// TwinCAT 3 PLC project EngineeringToolbox
// Title: EngineeringToolbox
// Company: Beckhoff Electronics Mfg
// Author: Daniel Schlingmann
// ProjectVersion: 3.1.2.2
// Description: Engineering Toolbox Library The library is provided "as-is" for TwinCAT3.1 by the Beckhoff Industry Management for Electronics Manufacturing. Please check the function "DisclaimerStatement : WSTRING[1500]" in additon to the following disclaimer: THE SOFTWARE IS PROVIDED "AS IS", WITHOUT WARRANTY OF ANY KIND, EXPRESS OR IMPLIED, INCLUDING BUT NOT LIMITED TO THE WARRANTIES OF MERCHANTABILITY, FITNESS FOR A PARTICULAR PURPOSE AND NONINFRINGEMENT. IN NO EVENT SHALL THE AUTHORS OR COPYRIGHT HOLDERS BE LIABLE FOR ANY CLAIM, DAMAGES OR OTHER LIABILITY, WHETHER IN AN ACTION OF CONTRACT, TORT OR OTHERWISE, ARISING FROM, OUT OF OR IN CONNECTION WITH THE SOFTWARE OR THE USE OR OTHER DEALINGS IN THE SOFTWARE.
// ProgramVersion: 3.1.4022.7
// libraries:
//   Tc2_Drive, * (Beckhoff Automation GmbH)
//   Tc2_EtherCAT, * (Beckhoff Automation GmbH)
//   Tc2_IoFunctions, * (Beckhoff Automation GmbH)
//   Tc2_Math, * (Beckhoff Automation GmbH)
//   Tc2_MC2, * (Beckhoff Automation GmbH)
//   Tc2_MC2_Camming, * (Beckhoff Automation GmbH)
//   Tc2_MC2_Drive, * (Beckhoff Automation GmbH)
//   Tc2_MC2_FlyingSaw, * (Beckhoff Automation GmbH)
//   Tc2_MDP, * (Beckhoff Automation GmbH)
//   Tc2_ModbusRTU, * (Beckhoff Automation GmbH)
//   Tc2_ModbusSrv, * (Beckhoff Automation GmbH)
//   Tc2_NC, * (Beckhoff Automation GmbH)
//   Tc2_NCI, * (Beckhoff Automation GmbH)
//   Tc2_NcKinematicTransformation, * (Beckhoff Automation GmbH)
//   Tc2_PlcInterpolation, * (Beckhoff Automation GmbH)
//   Tc2_SerialCom, * (Beckhoff Automation GmbH)
//   Tc2_Smtp, * (Beckhoff Automation GmbH)
//   Tc2_Standard, * (Beckhoff Automation GmbH)
//   Tc2_SUPS, * (Beckhoff Automation GmbH)
//   Tc2_System, * (Beckhoff Automation GmbH)
//   Tc2_TcpIp, * (Beckhoff Automation GmbH)
//   Tc2_Utilities, * (Beckhoff Automation GmbH)
//   Tc2_XmlDataSrv, * (Beckhoff Automation GmbH)
//   Tc3_Module, * (Beckhoff Automation GmbH)
//   Tc2_BackupRestoreEL6900,newest,Beckhoff Automation GmbH
// project tree:
//   GVLs/ Gvl.TcGVL (not stored), PARAM.TcGVL (not stored)
//   POUs/BoundsCheck/ boundsError.TcPOU (not stored), boundsOK.TcPOU (not stored), checkBounds.TcPOU (not stored), CheckBoundsInfo.TcPOU (not stored)
//   POUs/Connectivity/ADS/ AdsDataExchange.TcPOU
//   POUs/Connectivity/ Ipv4Addr_TO_UDINT.TcPOU, U_DEVICE_COM_CACHE.TcDUT (not stored), U_IPv4Addr.TcDUT (not stored), isValidIPv4Addr.TcPOU (not stored)
//   POUs/Connectivity/TF6310-TcpServer/DeviceCom/ TCPDeviceCom_SendRecBytes.TcPOU (not stored), TCPDeviceCom_SendRecString.TcPOU (not stored)
//   POUs/Connectivity/TF6340-SerialCom/ComPortDeviceCom/ ComPortDeviceCom_BufferHandle.TcPOU (not stored), ComPortDeviceCom_SendRecBytes.TcPOU (not stored), ComPortDeviceCom_SendRecString.TcPOU (not stored), ComPortEL6x22BEasyConnect.TcPOU (not stored)
//   POUs/Connectivity/TF6340-SerialCom/ComPortBasic/ ComPortBackground.TcPOU (not stored), ComPortSendRec.TcPOU (not stored)
//   POUs/Connectivity/TF625x-Modbus/Master/TF6250-ModbusTcpServer/TCP/ ModbusTcpMaster.TcPOU (not stored)
//   POUs/Connectivity/TF625x-Modbus/Master/TF6250-ModbusTcpServer/UDP/ ModbusUdpMaster.TcPOU
//   POUs/Connectivity/TF625x-Modbus/Master/TF6255-ModbusRtu/ ModbusRtuMaster22B.TcPOU (not stored), ModbusRtuMaster5B.TcPOU (not stored), ModbusRtuMasterPC.TcPOU
//   POUs/Connectivity/TF625x-Modbus/Master/_Components/ ModbusJob.TcPOU (not stored), ModbusSlaveCom.TcPOU (not stored)
//   POUs/Connectivity/TF625x-Modbus/Slave/ ModbusSlaveBase.TcPOU (not stored)
//   POUs/Connectivity/TF6310-TcpServer/TcpBasic/ TCPSendRecCtrl.TcPOU (not stored), TCPConnectionCtrl.TcPOU (not stored), TCPSocketCtrl.TcPOU (not stored)
//   POUs/Connectivity/TF6310-TcpServer/UdpBasic/ UDPSendRecCtrl.TcPOU, UDPServerCtrl.TcPOU (not stored), UDPSocketCtrl.TcPOU (not stored)
//   POUs/ControllerTools/ AverageFilter.TcPOU (not stored), PIDController.TcPOU (not stored), PT1Filter.TcPOU, signum.TcPOU (not stored), SlewRateLimitter.TcPOU (not stored), SlidingAverageExt.TcPOU (not stored), SlidingAverage.TcPOU (not stored), ThreePointController.TcPOU (not stored)
//   POUs/DataBuffer/ DoubleBuffer.TcPOU (not stored), Quicksort.TcPOU (not stored)
//   POUs/DataBuffer/Fifo/ Fifo.TcPOU (not stored), FifoExt.TcPOU (not stored), FifoLRealSimple.TcPOU (not stored), FifoBase.TcPOU (not stored)
//   POUs/DataBuffer/Ringbuffer/ RingbufferBase.TcPOU (not stored), Ringbuffer.TcPOU (not stored), RingbufferCharSimple.TcPOU (not stored), RingbufferExt.TcPOU, RingbufferByteSimple.TcPOU (not stored), RingbufferLRealSimple.TcPOU (not stored)
//   POUs/EventLogger/ EventsWriteToLogbook.TcPOU (not stored), EVENT_HANDLING_CONFIG.TcDUT (not stored), getEventClassPriority.TcPOU, getEventClassText.TcPOU (not stored), SOURCE_ID.TcDUT (not stored)
//   POUs/EventLogger/ReadEvents/ EventlogRead.TcPOU (not stored), EVENTLOG_READ_DATA.TcDUT (not stored), EVENTLOG_READ_HANDLEINFO.TcDUT (not stored), EVENTLOG_READ_STREAM.TcDUT, EVENTLOG_READ_STREAM_DATA_RAW.TcDUT (not stored), EVENTLOG_READ_STREAM_DATA_RAW_EX.TcDUT (not stored)
//   POUs/EventLogger/TriggerEvents/ EventHandling.TcPOU (not stored), EventHandlingGrp10.TcPOU (not stored), EventHandlingGrp25.TcPOU (not stored), EventHandlingGrp50.TcPOU (not stored), EventHandlingGrpCustomized.TcPOU (not stored), EventHandlingConfirmIsReq.TcPOU (not stored), EventHandlingStatisticInfo.TcPOU (not stored)
//   POUs/Fieldbus/CANopen/ CANopenMasterDiag.TcPOU (not stored), CANopenMasterIO.TcPOU (not stored)
//   POUs/Fieldbus/EAP/ EAP_PUB_SUB_IO.TcPOU (not stored), EAP_DEVICE_IO.TcPOU (not stored), EAP_PUB_VAR.TcPOU (not stored), EAP_SUB_VAR.TcPOU (not stored)
//   POUs/Fieldbus/EtherCAT/ EcCoEReadNewestDiagMsg.TcPOU (not stored), EcDiagBase.TcPOU (not stored), EcDiagBase_wEvents.TcPOU (not stored)
//   POUs/Fieldbus/EtherCAT/_Components/ EcMasterIO.TcPOU (not stored), EcMasterSupervisor.TcPOU (not stored), EcSlavesDiag.TcPOU (not stored), EcSlaveSupervisor.TcPOU (not stored), EC_MASTER_DEVICE_STATE.TcDUT (not stored), EC_SLAVE_DIAG_INFO_DATA.TcDUT (not stored)
//   POUs/Fieldbus/Profibus/ ProfibusMasterDiag.TcPOU, ProfibusMasterIO.TcPOU (not stored)
//   POUs/Fieldbus/Profinet/ ProfinetControllerIO.TcPOU (not stored), ProfinetControllerIO_wEvents.TcPOU, ProfinetDeviceIO.TcPOU
//   POUs/FileHandling/Basic/ FileHandling.TcPOU (not stored), ReadDirSimple.TcPOU (not stored), ReadDirSimpleExt.TcPOU (not stored)
//   POUs/FileHandling/TF6421-XmlServer/ XmlReadWrite.TcPOU (not stored), XmlReadWriteWithBackupFile.TcPOU (not stored)
//   POUs/IO/Analog/ AnalogIn.TcPOU, AnalogIn32.TcPOU, AnalogInELMBase.TcPOU (not stored), AnalogInELMSingleSampleDINT.TcPOU (not stored), AnalogInELMSingleSampleREAL.TcPOU (not stored), AnalogInREAL.TcPOU (not stored), AnalogOut.TcPOU
//   POUs/IO/ BlowOffSensors.TcPOU (not stored), Button.TcPOU (not stored), ButtonExt.TcPOU, Fuse.TcPOU (not stored), InOut.TcPOU (not stored), InOutExt.TcPOU, Input.TcPOU (not stored), Output.TcPOU (not stored)
//   POUs/IO/Cylinder/ Cylinder.TcPOU (not stored), CylinderExt.TcPOU (not stored), CylinderType4.TcPOU (not stored), I_Cylinder.TcIO (not stored)
//   POUs/IO/Drives/ AxDriveBase.TcPOU (not stored), AxDriveGetRef.TcPOU (not stored), I_AxDriveBase.TcIO (not stored)
//   POUs/IO/Drives/CoE/ AxDriveCoE.TcPOU (not stored), AxDriveCoE_wEvents.TcPOU (not stored), CiA_DS402Controlword.TcPOU (not stored), CiA_DS402Statusword.TcPOU (not stored), eCiA_DS402_CONTROL_CMD.TcDUT (not stored), eCiA_DS402_STATUS_STATE.TcDUT
//   POUs/IO/Drives/CoE/EL72xx/ AxDriveCoE_EL72xxParam.TcPOU (not stored), CiA_DS402StatuswordEx7xxx.TcPOU (not stored)
//   POUs/IO/Drives/DC/Ey73xx/ AxDriveDC.TcPOU (not stored), AxDriveDC_wEvents.TcPOU (not stored)
//   POUs/IO/Drives/SoE/ AxDriveSoE_Ax5000CommutationCalib.TcPOU (not stored), AxDriveSoE_Ax5000CalcPower.TcPOU (not stored), AxDriveSoE_Ax5000SwitchParamSet.TcPOU (not stored), Ax580x.TcPOU (not stored), AxDriveSoE_Ax5000.TcPOU (not stored), AxDriveSoE_Ax5000Param.TcPOU (not stored), AxDriveSoE_Ax5000wEvents.TcPOU (not stored), AxDriveSoE_Rexroth.TcPOU (not stored)
//   POUs/IO/Drives/SoE/Ax5000ParamSTRUCTs/P/ AX5000_P_0001.TcDUT (not stored), AX5000_P_0002.TcDUT (not stored), AX5000_P_0003.TcDUT (not stored), AX5000_P_0004.TcDUT (not stored), AX5000_P_0009.TcDUT (not stored), AX5000_P_0010.TcDUT (not stored), AX5000_P_0020.TcDUT (not stored), AX5000_P_0021.TcDUT (not stored), AX5000_P_0040.TcDUT (not stored), AX5000_P_0050.TcDUT (not stored), AX5000_P_0051.TcDUT (not stored), AX5000_P_0052.TcDUT (not stored), AX5000_P_0053.TcDUT (not stored), AX5000_P_0054.TcDUT (not stored), AX5000_P_0055.TcDUT (not stored), AX5000_P_0056.TcDUT (not stored), AX5000_P_0057.TcDUT (not stored), AX5000_P_0058.TcDUT, AX5000_P_0059.TcDUT (not stored), AX5000_P_0060.TcDUT (not stored), AX5000_P_0061.TcDUT (not stored), AX5000_P_0062.TcDUT (not stored), AX5000_P_0063.TcDUT, AX5000_P_0064.TcDUT (not stored), AX5000_P_0065.TcDUT (not stored), AX5000_P_0066.TcDUT (not stored), AX5000_P_0067.TcDUT (not stored), AX5000_P_0068.TcDUT (not stored), AX5000_P_0069.TcDUT, AX5000_P_0070.TcDUT (not stored), AX5000_P_0071.TcDUT, AX5000_P_0072.TcDUT, AX5000_P_0073.TcDUT (not stored), AX5000_P_0074.TcDUT (not stored), AX5000_P_0075.TcDUT (not stored), AX5000_P_0076.TcDUT (not stored), AX5000_P_0077.TcDUT (not stored), AX5000_P_0078.TcDUT (not stored), AX5000_P_0088.TcDUT (not stored), AX5000_P_0089.TcDUT (not stored), AX5000_P_0090.TcDUT (not stored), AX5000_P_0091.TcDUT (not stored), AX5000_P_0092.TcDUT (not stored), AX5000_P_0093.TcDUT (not stored), AX5000_P_0096.TcDUT (not stored), AX5000_P_0097.TcDUT (not stored), AX5000_P_0098_beckhoff.TcDUT (not stored), AX5000_P_0098_beckhoff_electrical_data.TcDUT (not stored), AX5000_P_0099.TcDUT (not stored), AX5000_P_0100.TcDUT (not stored), AX5000_P_0101.TcDUT (not stored), AX5000_P_0102.TcDUT (not stored), AX5000_P_0103.TcDUT (not stored), AX5000_P_0104.TcDUT (not stored), AX5000_P_0105.TcDUT (not stored), AX5000_P_0106.TcDUT, AX5000_P_0107.TcDUT (not stored), AX5000_P_0108.TcDUT (not stored), AX5000_P_0109.TcDUT (not stored), AX5000_P_0110.TcDUT (not stored), AX5000_P_0111.TcDUT (not stored), AX5000_P_0112.TcDUT (not stored), AX5000_P_0113.TcDUT (not stored), AX5000_P_0114.TcDUT (not stored), AX5000_P_0115.TcDUT (not stored), AX5000_P_0116.TcDUT (not stored), AX5000_P_0117.TcDUT (not stored), AX5000_P_0118.TcDUT (not stored), AX5000_P_0119.TcDUT (not stored), AX5000_P_0125.TcDUT, AX5000_P_0126.TcDUT (not stored), AX5000_P_0127.TcDUT, AX5000_P_0128.TcDUT (not stored), AX5000_P_0150.TcDUT (not stored), AX5000_P_0151.TcDUT (not stored), AX5000_P_0152.TcDUT (not stored), AX5000_P_0153.TcDUT (not stored), AX5000_P_0154.TcDUT (not stored), AX5000_P_0155.TcDUT (not stored), AX5000_P_0158.TcDUT (not stored), AX5000_P_0159.TcDUT (not stored), AX5000_P_0160.TcDUT (not stored), AX5000_P_0161.TcDUT (not stored), AX5000_P_0162.TcDUT (not stored), AX5000_P_0163.TcDUT (not stored), AX5000_P_0165.TcDUT (not stored), AX5000_P_0166.TcDUT (not stored), AX5000_P_0167.TcDUT (not stored), AX5000_P_0168.TcDUT (not stored), AX5000_P_0169.TcDUT (not stored), AX5000_P_0170.TcDUT, AX5000_P_0171.TcDUT (not stored), AX5000_P_0180.TcDUT (not stored), AX5000_P_0181.TcDUT, AX5000_P_0182.TcDUT (not stored), AX5000_P_0183.TcDUT (not stored), AX5000_P_0184.TcDUT (not stored), AX5000_P_0185.TcDUT (not stored), AX5000_P_0188.TcDUT (not stored), AX5000_P_0189.TcDUT (not stored), AX5000_P_0192.TcDUT (not stored), AX5000_P_0193.TcDUT (not stored), AX5000_P_0196.TcDUT (not stored), AX5000_P_0198.TcDUT, AX5000_P_0199.TcDUT (not stored), AX5000_P_0200.TcDUT, AX5000_P_0201.TcDUT (not stored), AX5000_P_0202.TcDUT, AX5000_P_0203.TcDUT (not stored), AX5000_P_0204.TcDUT (not stored), AX5000_P_0205.TcDUT (not stored), AX5000_P_0206.TcDUT, AX5000_P_0207.TcDUT, AX5000_P_0208.TcDUT, AX5000_P_0209.TcDUT, AX5000_P_0210.TcDUT (not stored), AX5000_P_0211.TcDUT, AX5000_P_0212.TcDUT (not stored), AX5000_P_0213.TcDUT (not stored), AX5000_P_0214.TcDUT (not stored), AX5000_P_0215.TcDUT (not stored), AX5000_P_0216.TcDUT (not stored), AX5000_P_0217.TcDUT, AX5000_P_0218.TcDUT (not stored), AX5000_P_0219.TcDUT (not stored), AX5000_P_0220.TcDUT (not stored), AX5000_P_0221.TcDUT (not stored), AX5000_P_0250.TcDUT (not stored), AX5000_P_0251.TcDUT (not stored), AX5000_P_0252.TcDUT (not stored), AX5000_P_0253.TcDUT (not stored), AX5000_P_0254.TcDUT, AX5000_P_0255.TcDUT (not stored), AX5000_P_0256.TcDUT (not stored), AX5000_P_0270.TcDUT (not stored), AX5000_P_0271.TcDUT (not stored), AX5000_P_0272.TcDUT (not stored), AX5000_P_0273.TcDUT (not stored), AX5000_P_0274.TcDUT (not stored), AX5000_P_0275.TcDUT (not stored), AX5000_P_0276.TcDUT (not stored), AX5000_P_0277.TcDUT (not stored), AX5000_P_0278.TcDUT (not stored), AX5000_P_0300.TcDUT (not stored), AX5000_P_0301.TcDUT (not stored), AX5000_P_0302.TcDUT, AX5000_P_0303.TcDUT (not stored), AX5000_P_0304.TcDUT (not stored), AX5000_P_0305.TcDUT (not stored), AX5000_P_0306.TcDUT (not stored), AX5000_P_0307.TcDUT (not stored), AX5000_P_0308.TcDUT (not stored), AX5000_P_0309.TcDUT (not stored), AX5000_P_0310.TcDUT (not stored), AX5000_P_0311.TcDUT (not stored), AX5000_P_0312.TcDUT (not stored), AX5000_P_0313.TcDUT (not stored), AX5000_P_0314.TcDUT (not stored), AX5000_P_0315.TcDUT (not stored), AX5000_P_0316.TcDUT (not stored), AX5000_P_0317.TcDUT (not stored), AX5000_P_0320.TcDUT (not stored), AX5000_P_0321.TcDUT (not stored), AX5000_P_0322.TcDUT (not stored), AX5000_P_0323.TcDUT (not stored), AX5000_P_0324.TcDUT (not stored), AX5000_P_0325.TcDUT (not stored), AX5000_P_0326.TcDUT (not stored), AX5000_P_0350.TcDUT (not stored), AX5000_P_0351.TcDUT (not stored), AX5000_P_0352.TcDUT, AX5000_P_0353.TcDUT (not stored), AX5000_P_0354.TcDUT, AX5000_P_0356.TcDUT (not stored), AX5000_P_0360.TcDUT (not stored), AX5000_P_0361.TcDUT (not stored), AX5000_P_0400.TcDUT (not stored), AX5000_P_0401.TcDUT (not stored), AX5000_P_0402.TcDUT (not stored), AX5000_P_0451.TcDUT (not stored), AX5000_P_0452.TcDUT (not stored), AX5000_P_0453.TcDUT (not stored), AX5000_P_0454.TcDUT (not stored), AX5000_P_0455.TcDUT (not stored), AX5000_P_0456.TcDUT (not stored), AX5000_P_0457.TcDUT (not stored), AX5000_P_0458.TcDUT (not stored), AX5000_P_0459.TcDUT (not stored), AX5000_P_0460.TcDUT (not stored), AX5000_P_0461.TcDUT (not stored), AX5000_P_0462.TcDUT (not stored), AX5000_P_0463.TcDUT (not stored), AX5000_P_0464.TcDUT, AX5000_P_0502.TcDUT (not stored), AX5000_P_0503.TcDUT (not stored), AX5000_P_0504.TcDUT (not stored), AX5000_P_0505.TcDUT, AX5000_P_0511.TcDUT (not stored), AX5000_P_0512.TcDUT (not stored), AX5000_P_0513.TcDUT (not stored), AX5000_P_0514.TcDUT, AX5000_P_0515.TcDUT (not stored), AX5000_P_0516.TcDUT, AX5000_P_0517.TcDUT (not stored), AX5000_P_0518.TcDUT (not stored), AX5000_P_0552.TcDUT (not stored), AX5000_P_0553.TcDUT (not stored), AX5000_P_0554.TcDUT (not stored), AX5000_P_0555.TcDUT (not stored), AX5000_P_0556.TcDUT (not stored), AX5000_P_0557.TcDUT, AX5000_P_0558.TcDUT (not stored), AX5000_P_0601.TcDUT (not stored), AX5000_P_0602.TcDUT (not stored), AX5000_P_0610.TcDUT (not stored), AX5000_P_0611.TcDUT (not stored), AX5000_P_0800.TcDUT (not stored), AX5000_P_0801.TcDUT (not stored), AX5000_P_0802.TcDUT (not stored), AX5000_P_0804.TcDUT (not stored), AX5000_P_0805.TcDUT (not stored), AX5000_P_0806.TcDUT (not stored), AX5000_P_0810.TcDUT (not stored), AX5000_P_0811.TcDUT, AX5000_P_0850.TcDUT (not stored), AX5000_P_0851.TcDUT (not stored), AX5000_P_0900.TcDUT, AX5000_P_0901.TcDUT (not stored), AX5000_P_0902.TcDUT (not stored), AX5000_P_0904.TcDUT (not stored), AX5000_P_0905.TcDUT (not stored), AX5000_P_0906.TcDUT (not stored), AX5000_P_0912.TcDUT (not stored), AX5000_P_1000.TcDUT (not stored), AX5000_P_1001.TcDUT (not stored), AX5000_P_1002.TcDUT (not stored), AX5000_P_1003.TcDUT (not stored), AX5000_P_1004.TcDUT (not stored), AX5000_P_1005.TcDUT (not stored), AX5000_P_1006.TcDUT (not stored), AX5000_P_1007.TcDUT (not stored), AX5000_P_1008.TcDUT (not stored), AX5000_P_1009.TcDUT, AX5000_P_1010.TcDUT, AX5000_P_1011.TcDUT (not stored), AX5000_P_1012.TcDUT (not stored), AX5000_P_1020.TcDUT (not stored), AX5000_P_1021.TcDUT (not stored), AX5000_P_1022.TcDUT (not stored), AX5000_P_2000.TcDUT (not stored), AX5000_P_2001.TcDUT (not stored), AX5000_P_2002.TcDUT (not stored)
//   POUs/IO/Drives/SoE/Ax5000ParamSTRUCTs/S/ AX5000_S_0001.TcDUT (not stored), AX5000_S_0002.TcDUT (not stored), AX5000_S_0007.TcDUT (not stored), AX5000_S_0011.TcDUT (not stored), AX5000_S_0012.TcDUT (not stored), AX5000_S_0013.TcDUT (not stored), AX5000_S_0015.TcDUT (not stored), AX5000_S_0016.TcDUT, AX5000_S_0017.TcDUT (not stored), AX5000_S_0018.TcDUT (not stored), AX5000_S_0024.TcDUT, AX5000_S_0029.TcDUT, AX5000_S_0030.TcDUT (not stored), AX5000_S_0031.TcDUT (not stored), AX5000_S_0032.TcDUT, AX5000_S_0033.TcDUT (not stored), AX5000_S_0034.TcDUT (not stored), AX5000_S_0035.TcDUT, AX5000_S_0036.TcDUT, AX5000_S_0037.TcDUT (not stored), AX5000_S_0040.TcDUT (not stored), AX5000_S_0043.TcDUT (not stored), AX5000_S_0044.TcDUT (not stored), AX5000_S_0045.TcDUT (not stored), AX5000_S_0046.TcDUT (not stored), AX5000_S_0047.TcDUT (not stored), AX5000_S_0048.TcDUT (not stored), AX5000_S_0051.TcDUT (not stored), AX5000_S_0053.TcDUT (not stored), AX5000_S_0055.TcDUT, AX5000_S_0076.TcDUT (not stored), AX5000_S_0079.TcDUT (not stored), AX5000_S_0080.TcDUT (not stored), AX5000_S_0081.TcDUT (not stored), AX5000_S_0082.TcDUT, AX5000_S_0083.TcDUT, AX5000_S_0084.TcDUT (not stored), AX5000_S_0085.TcDUT (not stored), AX5000_S_0086.TcDUT (not stored), AX5000_S_0091.TcDUT (not stored), AX5000_S_0092.TcDUT (not stored), AX5000_S_0095.TcDUT (not stored), AX5000_S_0099.TcDUT (not stored), AX5000_S_0100.TcDUT (not stored), AX5000_S_0101.TcDUT (not stored), AX5000_S_0103.TcDUT (not stored), AX5000_S_0104.TcDUT (not stored), AX5000_S_0106.TcDUT (not stored), AX5000_S_0107.TcDUT (not stored), AX5000_S_0109.TcDUT (not stored), AX5000_S_0110.TcDUT (not stored), AX5000_S_0111.TcDUT (not stored), AX5000_S_0112.TcDUT, AX5000_S_0113.TcDUT (not stored), AX5000_S_0119.TcDUT (not stored), AX5000_S_0120.TcDUT (not stored), AX5000_S_0124.TcDUT (not stored), AX5000_S_0126.TcDUT (not stored), AX5000_S_0130.TcDUT (not stored), AX5000_S_0131.TcDUT (not stored), AX5000_S_0134.TcDUT (not stored), AX5000_S_0135.TcDUT (not stored), AX5000_S_0136.TcDUT (not stored), AX5000_S_0137.TcDUT (not stored), AX5000_S_0143.TcDUT (not stored), AX5000_S_0149.TcDUT (not stored), AX5000_S_0159.TcDUT (not stored), AX5000_S_0160.TcDUT (not stored), AX5000_S_0161.TcDUT (not stored), AX5000_S_0162.TcDUT (not stored), AX5000_S_0163.TcDUT (not stored), AX5000_S_0169.TcDUT (not stored), AX5000_S_0170.TcDUT (not stored), AX5000_S_0179.TcDUT (not stored), AX5000_S_0185.TcDUT (not stored), AX5000_S_0186.TcDUT (not stored), AX5000_S_0187.TcDUT (not stored), AX5000_S_0188.TcDUT (not stored), AX5000_S_0189.TcDUT (not stored), AX5000_S_0196.TcDUT (not stored), AX5000_S_0200.TcDUT (not stored), AX5000_S_0201.TcDUT (not stored), AX5000_S_0203.TcDUT (not stored), AX5000_S_0204.TcDUT (not stored), AX5000_S_0206.TcDUT (not stored), AX5000_S_0207.TcDUT (not stored), AX5000_S_0216.TcDUT (not stored), AX5000_S_0217.TcDUT (not stored), AX5000_S_0219.TcDUT (not stored), AX5000_S_0254.TcDUT (not stored), AX5000_S_0256.TcDUT (not stored), AX5000_S_0257.TcDUT (not stored), AX5000_S_0267.TcDUT (not stored), AX5000_S_0273.TcDUT (not stored), AX5000_S_0274.TcDUT (not stored), AX5000_S_0292.TcDUT (not stored), AX5000_S_0295.TcDUT, AX5000_S_0296.TcDUT (not stored), AX5000_S_0347.TcDUT (not stored), AX5000_S_0348.TcDUT, AX5000_S_0372.TcDUT (not stored), AX5000_S_0374.TcDUT (not stored), AX5000_S_0375.TcDUT (not stored), AX5000_S_0380.TcDUT (not stored), AX5000_S_0381.TcDUT (not stored), AX5000_S_0383.TcDUT (not stored), AX5000_S_0384.TcDUT (not stored), AX5000_S_0390.TcDUT (not stored), AX5000_S_0403.TcDUT (not stored), AX5000_S_0405.TcDUT (not stored), AX5000_S_0409.TcDUT (not stored), AX5000_S_0410.TcDUT (not stored), AX5000_S_0429.TcDUT (not stored), AX5000_S_0432.TcDUT (not stored), AX5000_S_0435.TcDUT (not stored), AX5000_S_0436.TcDUT (not stored)
//   POUs/IO/Drives/Stepper/ AxDriveStepper.TcPOU (not stored), AxDriveStepperParam.TcPOU (not stored), AxDriveStepper_wEvents.TcPOU
//   POUs/IO/EL-EP/ AnalogOut_EL2535.TcPOU, EL1262_Base.TcPOU (not stored), EL3681.TcPOU, EL1904.TcPOU, EL69xx.TcPOU (not stored), EL3356.TcPOU (not stored), Eyx9xx.TcPOU (not stored), ZB8610.TcPOU (not stored)
//   POUs/IO/EL-EP/EL9x/ EL9501.TcPOU (not stored), EL9576.TcPOU (not stored), EL95xxPowerTerminal.TcPOU (not stored), ELSystemTerminal.TcPOU (not stored)
//   POUs/IO/_EcSlaveFWUpdater/ EcSlaveDevFWUpdater.TcPOU
//   POUs/IO/_EcSlaveInfoDataIO/ EcSlaveInfoData.TcPOU, EcSlaveInfoDataExt.TcPOU (not stored), I_EcSlaveInfoData.TcIO (not stored)
//   POUs/IO/EL-EP/EL3403/ EL3403.TcPOU, EL3403Logic.TcPOU (not stored)
//   POUs/IO/EL-EP/EP92xxPwrBox/ EP9214.TcPOU (not stored), EP9214_CHANNEL.TcPOU (not stored), EP9224_0037.TcPOU (not stored), EP9224_0037_CHANNEL.TcPOU (not stored)
//   POUs/IO/FreqConv/EtherCAT/DS402/ EcFcDS402_ComBase.TcPOU (not stored)
//   POUs/IO/FreqConv/ IOFcCom.TcPOU (not stored)
//   POUs/IO/Motors/ IOMotor.TcPOU (not stored), IOMotor2Dir.TcPOU, IOMotorStarDelta.TcPOU
//   POUs/IO/[underDev]/ Cylinder_wUnitItf.TcPOU (not stored)
//   POUs/IO/_ItfActuators/ I_ActuatorBase.TcIO (not stored), I_ActuatorEnableDisable.TcIO (not stored), I_ActuatorFwdRev.TcIO (not stored), I_ActuatorFwdBwd.TcIO (not stored), I_ActuatorLeftRight.TcIO (not stored), I_ActuatorOnOff.TcIO (not stored), I_ActuatorOpenClose.TcIO (not stored), I_ActuatorPosNeg.TcIO, I_ActuatorStartStop.TcIO (not stored), I_ActuatorUpDown.TcIO, I_ActuatorWorkBase.TcIO (not stored)
//   POUs/IpcDiag/MDP/InfoModuls/ MDP_CPU.TcPOU (not stored), MDP_Fan.TcPOU (not stored), MDP_Mainboard.TcPOU (not stored), MDP_RaidSimple.TcPOU, MDP_ReadModulList.TcPOU (not stored), MDP_SiliconDrives.TcPOU (not stored), MDP_UPS.TcPOU (not stored)
//   POUs/IpcDiag/MDP/ MDP_Info.TcPOU (not stored), MDP_IpcDiag.TcPOU (not stored), MDP_IpcDiag_wEvents.TcPOU (not stored)
//   POUs/IpcDiag/ UPSStatus.TcPOU (not stored)
//   POUs/Logging/ DataFileLogger.TcPOU (not stored), DataUdpLogger.TcPOU (not stored), I_LogbookSubscriber.TcIO, I_Logbook.TcIO (not stored), Logbook.TcPOU, LogbookData.TcDUT (not stored), LogbookPuplisher.TcPOU (not stored), LogbookSubEventLog.TcPOU (not stored), LogbookSubSendMail.TcPOU (not stored), adsLogError.TcPOU (not stored), adsLogHint.TcPOU (not stored), adsLogWarn.TcPOU (not stored), LogbookSubSysLog.TcPOU (not stored), LogbookSubWriteFile.TcPOU (not stored), Logbook_wEventClass.TcPOU (not stored), adsLogwTcEventClass.TcPOU (not stored)
//   POUs/Motion/TF50xx-NC/00_Base/ I_AxNcPTP.TcIO (not stored), AxFbBase.TcPOU (not stored), AxRWParaBase.TcPOU (not stored), I_AxNcBase.TcIO (not stored)
//   POUs/Motion/TF50xx-NC/02_Options/Parameter/ AxPara.TcPOU (not stored), AxParaCtrl.TcPOU (not stored)
//   POUs/Motion/TF50xx-NC/03_Utilities/ AxAutoWriteSoftLimit.TcPOU (not stored), CoordinateTransformation2D.TcPOU, AxCalcPosBias.TcPOU (not stored), AxResonanceAvoidance.TcPOU (not stored) (excluded from build), AxSoftSyncDistance.TcPOU (not stored), AxStatemodel.TcPOU, AxAutoFct.TcPOU (not stored), AX_JOB.TcPOU (not stored), getOvrVelo.TcPOU (not stored)
//   POUs/Motion/TF50xx-NC/ AxNcPTPwJobs.TcPOU, AxNcBaseExt.TcPOU, AxNcPtpGear.TcPOU (not stored), AxNcBase.TcPOU (not stored), AxNcPTP.TcPOU (not stored)
//   POUs/Motion/TF5100-NCI/ NciChannel_wEvents.TcPOU (not stored), NciChannel.TcPOU (not stored)
//   POUs/Motion/TF511x-KIN/03_DUTs/Positions/ KIN_POSITIONS.TcPOU (not stored), KIN_POSITIONS_ACS_DUT.TcDUT (not stored), KIN_POSITIONS_MCS_DUT.TcDUT (not stored), U_KIN_POSITIONS.TcDUT (not stored)
//   POUs/Motion/TF511x-KIN/03_DUTs/Trafo/ KIN_CALCTRAFO_AXPOS_PARAM.TcPOU (not stored), KIN_STATE_OBSERVER_OID_PARAM.TcPOU (not stored), KIN_STATICTRAFO_PARAM.TcPOU, KIN_TOOLTRAFO_PARAM.TcPOU (not stored), UCS.TcPOU
//   POUs/Motion/ VALUE_3D.TcPOU, VALUE_3D_DUT.TcDUT (not stored), VALUE_6D.TcPOU (not stored), VALUE_6D_DUT.TcDUT (not stored)
//   POUs/Safety/Diag/ SafetyLogicAndIOTerminalDiag.TcPOU, SafetyIODeviceDiagRead.TcPOU (not stored), SafetyIODeviceDiag_wEvents.TcPOU (not stored), SafetyIOsDiag.TcPOU (not stored), SafetyLogicTerminalDiag.TcPOU (not stored), SafetyPlcTerminalDiag.TcPOU (not stored)
//   POUs/StringHelper/ cutStrNumberToSeperator.TcPOU (not stored), replaceUmlauts.TcPOU (not stored), cutStrToSeperator.TcPOU (not stored), cutWStrToSeperator.TcPOU, DWORD_TO_BINSTR_EXT.TcPOU (not stored), DWORD_TO_HEXSTR_EXT.TcPOU (not stored), getCntCharInStr.TcPOU (not stored), getCntCharInWStr.TcPOU (not stored), isWStringNumeric.TcPOU (not stored), HEXSTR_TO_DWORD.TcPOU (not stored), HEXSTR_TO_LWORD.TcPOU (not stored), INSERT_EXT.TcPOU (not stored), LWORD_TO_BINSTR_EXT.TcPOU (not stored), LWORD_TO_HEXSTR_EXT.TcPOU (not stored), readStrToSeperator.TcPOU (not stored), replaceInString.TcPOU (not stored), getFilledString.TcPOU, isStringNumeric.TcPOU (not stored), readWStrToSeperator.TcPOU, replaceInWString.TcPOU (not stored), U_MAX_STRING.TcDUT (not stored), U_MAX_WSTRING.TcDUT (not stored), WINSERT_EXT.TcPOU (not stored)
//   POUs/System/ SystemInfo.TcPOU (not stored), SystemInfo64.TcPOU (not stored) (excluded from build), SystemPulses.TcPOU (not stored), TaskInfo.TcPOU (not stored)
//   POUs/TimeHelper/ PartsPerTime.TcPOU (not stored), createTOD.TcPOU (not stored), getDateAndTimeDelta.TcPOU (not stored), getTonCountdown.TcPOU (not stored), LivebitCheck.TcPOU (not stored), Ontime.TcPOU (not stored), OntimeExt.TcPOU (not stored), OntimeSimple.TcPOU (not stored), Pulse.TcPOU (not stored), SensorTimeoutCheck.TcPOU (not stored), systemtimeInCam.TcPOU (not stored), systemtimeCmp.TcPOU (not stored), systemtimeInWin.TcPOU (not stored), TimeSwitch.TcPOU (not stored), TONRecord.TcPOU, TONTOF.TcPOU (not stored), VeloLinearMeasurement.TcPOU (not stored)
//   POUs/_Miscellaneous/64BitFunctions/ CLEARBIT64.TcPOU (not stored), CSETBIT64.TcPOU (not stored), GETBIT64.TcPOU (not stored), SETBIT64.TcPOU (not stored)
//   POUs/_Miscellaneous/ nextIdx.TcPOU (not stored), TC_VN_COLORS.TcDUT (not stored) (excluded from build), FbBase.TcPOU (not stored), CAM.TcPOU (not stored), CAM3D.TcPOU (not stored), COLOR.TcDUT (not stored), ERROR_HDL.TcPOU (not stored), FbBaseExt.TcPOU, FbBaseOutputs.TcPOU (not stored), getNoOfBits.TcPOU (not stored), LCID.TcDUT (not stored), eLCID.TcDUT (not stored), LOGx.TcPOU (not stored), OEECalculation.TcPOU (not stored), polynomial.TcPOU (not stored), RF_TRIG.TcPOU (not stored), scale.TcPOU, SEQUENCE_HDL.TcPOU (not stored), setNoOfBits.TcPOU (not stored), TEST_FB.TcPOU, TOGGLE.TcPOU (not stored), U_32BIT_DATATYPE.TcDUT (not stored), U_64BIT_DATATYPE.TcDUT (not stored), WIN.TcPOU (not stored)
//   POUs/_Miscellaneous/Conversions/ ADSERROR_TO_HRESULT.TcPOU (not stored), DWORD_TO_REAL_EX.TcPOU, HRESULT_TO_ADSERROR.TcPOU (not stored), REAL_TO_FMLREAL.TcPOU (not stored), LWORD_TO_LREAL_EX.TcPOU, SWAP_BYTES_OF_WORDS.TcPOU (not stored), SWAP_WORDS_OF_DWORD.TcPOU (not stored), SWAP_WORDS_OF_LWORD.TcPOU (not stored), ADSERROR_TO_WIN32ERROR.TcPOU (not stored), ADSERROR_TO_WSERROR.TcPOU (not stored), C_TO_F.TcPOU (not stored), DEGREES_TO_RPM.TcPOU (not stored), F_TO_C.TcPOU (not stored), GF_TO_N.TcPOU (not stored), TO_FMLREAL.TcPOU, MMIN_TO_MMS.TcPOU (not stored), MMS_TO_MMIN.TcPOU (not stored), N_TO_GF.TcPOU (not stored), RPM_TO_DEGREES.TcPOU (not stored)
//   POUs/Safety/ SafetyCircuit.TcPOU (not stored), SafetyGroupIO.TcPOU (not stored), SafetyPlcBackupRestore.TcPOU (not stored), SAFETY_CIRCUIT_STATUS.TcDUT (not stored)
//   POUs/Statemodel/control/ I_StatemodelBase.TcIO (not stored), I_Statemodel.TcIO (not stored), Statemodel.TcPOU (not stored)
//   POUs/Statemodel/ eMODE.TcDUT (not stored), eSTATE.TcDUT (not stored)
//   POUs/Statemodel/UnitTemplate/ I_Statemodel_Unit.TcIO (not stored), Statemodel_Unit.TcPOU (not stored)
//   POUs/Motion/TF50xx-NC/01_Main/ AxAdmin.TcPOU (not stored), AxHoming.TcPOU (not stored), AxMotion.TcPOU (not stored)
//   POUs/Motion/TF50xx-NC/02_Options/Motion/ AxSuperposition.TcPOU (not stored), AxMoveSinus.TcPOU (not stored), AxHomingOnBlock.TcPOU (not stored)
//   POUs/Motion/TF5100-NCI/01_Main/ NciAdmin.TcPOU (not stored), NciGrp.TcPOU (not stored), NciItp.TcPOU, NciMotion.TcPOU, NCI_REF.TcPOU (not stored)
//   POUs/Motion/TF5100-NCI/02_Options/Error/ NciChnEventHandling.TcPOU (not stored), NciEventHandling.TcPOU (not stored)
//   POUs/Motion/TF5100-NCI/02_Options/MFunctions/ NciMFnc.TcPOU (not stored)
//   POUs/Motion/TF5100-NCI/02_Options/PlcItp/ NciCreateItpTable.TcPOU (not stored), NciCreateItpTableEntryTemplate.TcPOU
//   POUs/Motion/TF5100-NCI/02_Options/RParameter/ NCiReadWriteRParam.TcPOU (not stored)
//   POUs/Motion/TF511x-KIN/01_Main/ KinAdmin.TcPOU (not stored), KIN_REF.TcPOU (not stored)
//   POUs/Motion/TF511x-KIN/02_Options/ KinLockUnlockTrafoParam.TcPOU (not stored), KinWriteToolTrafoParam.TcPOU (not stored), KinWriteUCSTrafoParam.TcPOU
//   POUs/Motion/TF511x-KIN/ KinChannel.TcPOU (not stored)
//   POUs/Motion/TF50xx-NC/02_Options/Coupling/ AxCamming.TcPOU (not stored), AxFlyingSaw.TcPOU (not stored), AxGear.TcPOU (not stored)
//   POUs/Motion/TF50xx-NC/02_Options/Error/ AxNcEventHandling.TcPOU (not stored), AxEventHandling.TcPOU
//   POUs/Motion/TF50xx-NC/02_Options/Phasing/ AxPhasing.TcPOU (not stored)
//   POUs/Motion/TF50xx-NC/02_Options/TouchProbe/ AxTouchProbe.TcPOU (not stored)
//   POUs/StringHelper/ExtendedString/ ExtString.TcPOU (not stored), ExtWString.TcPOU (not stored), T_EXT_STRING.TcDUT (not stored), T_EXT_WSTRING.TcDUT (not stored)
//   POUs/TimeHelper/Conversions/ FILETIME_TO_DATE.TcPOU (not stored), LREAL_TO_TIME_SEC.TcPOU (not stored), FILETIME_TO_TOD.TcPOU (not stored), SYSTEMTIME_TO_TIME.TcPOU (not stored), SYSTEMTIME_TO_TIME_EX.TcPOU (not stored), SYSTEMTIME_TO_TOD.TcPOU (not stored), SYSTEMTIME_TO_DATE.TcPOU (not stored), TIME_TO_FMRLREAL.TcPOU (not stored), TIME_TO_SYSTEMTIME.TcPOU (not stored)
//   Version/ disclaimerStatement.TcPOU (not stored), Global_Version.TcGVL (not stored)

// ---- POUs/EventLogger/ReadEvents/EVENTLOG_READ_STREAM.TcDUT
TYPE EVENTLOG_READ_STREAM :
STRUCT
	cbStream		: DWORD; //size OF this structure, including all following TcGetEventParams structures
	count			: DWORD;
	data			: EVENTLOG_READ_STREAM_DATA_RAW;	(* Stream OF TcGetEventParams *)
END_STRUCT
END_TYPE

// ---- POUs/IO/Drives/CoE/eCiA_DS402_STATUS_STATE.TcDUT
{attribute 'qualified_only'}
{attribute 'to_string'}
TYPE eCiA_DS402_STATUS_STATE :
(
	NOT_READY_TO_SWITCH_ON									:= 2#0000_0000, //2#x0xx_0000 / Not ready to switch on. The drive is initialising or being configured.
	SWITCH_ON_DISABLED										:= 2#0100_0000, //2#x1xx_0000 / The Drive will not accept a switch on command 
	READY_TO_SWITCH_ON										:= 2#0010_0001, //2#x01x_0001 / The Drive will accept a switch on command.
	SWITCHED_ON												:= 2#0010_0011, (* 2#x01x_0011 / The Drive will accept an Operation Enable (Run or Jog) command. 		
																				- Power stage of the Drive is ready to operate.
																				- Voltage has not yet been applied to the motor terminals*)
	OPERATION_ENABLED										:= 2#0010_0111,  (* 2#x01x_0111 / Normal operational state of the drive. This state includes Running, Jogging,
																				Stopping (Disabling Operation) and Shutting Down (Switching Off).
																				- Voltage applied to the motor terminals. *)
	QUICK_STOP_ACTIVE										:= 2#0000_0111, //2#x00x_0111 / Emergency stop (Fast stop) is active
    FAULT_REACTION_ACTIVE									:= 2#0000_1111, //2#x0xx_1111 / The Drive is processing a tripped event                                                                        
	FAULT_ACTIVE											:= 2#0000_1000 //2#x0xx_1000 / The Drive is in fault state and awaiting a reset trigger
	
);                                                                          
END_TYPE

// ---- POUs/IO/Drives/SoE/Ax5000ParamSTRUCTs/P/AX5000_P_0058.TcDUT
TYPE AX5000_P_0058 :
STRUCT
	Mechanical_commutation_offset:UINT;
END_STRUCT
END_TYPE

// ---- POUs/IO/Drives/SoE/Ax5000ParamSTRUCTs/P/AX5000_P_0063.TcDUT
TYPE AX5000_P_0063 :
STRUCT
	Thermal_motor_ulitisation:UINT;
END_STRUCT
END_TYPE

// ---- POUs/IO/Drives/SoE/Ax5000ParamSTRUCTs/P/AX5000_P_0069.TcDUT
TYPE AX5000_P_0069 :
STRUCT
	Actual_lenght:UINT:=2;
	Max_lenght:UINT:=2;
	velocity_limit:UINT:=100;
//	{attribute 'hide'}
	Rsvd:UINT;
END_STRUCT
END_TYPE

// ---- POUs/IO/Drives/SoE/Ax5000ParamSTRUCTs/P/AX5000_P_0071.TcDUT
TYPE AX5000_P_0071 :
STRUCT
	Actual_lenght:UINT;
	Max_lenght:UINT;
	Rotor_moment_of_inertia:UDINT;
	Load_moment_of_inertia:UDINT;
END_STRUCT
END_TYPE

// ---- POUs/IO/Drives/SoE/Ax5000ParamSTRUCTs/P/AX5000_P_0072.TcDUT
TYPE AX5000_P_0072 :
STRUCT
	Actual_lenght:UINT;
	Max_lenght:UINT;
	Holding_torque:UINT;
	Elektrical_power:UINT;
	Moment_of_inertia:UINT;
END_STRUCT
END_TYPE

// ---- POUs/IO/Drives/SoE/Ax5000ParamSTRUCTs/P/AX5000_P_0106.TcDUT
TYPE AX5000_P_0106 :
STRUCT
	ASM_connection_type:UINT;
END_STRUCT
END_TYPE

// ---- POUs/IO/Drives/SoE/Ax5000ParamSTRUCTs/P/AX5000_P_0125.TcDUT
TYPE AX5000_P_0125 :
STRUCT
	Pole_pair_distance:UINT;
END_STRUCT
END_TYPE

// ---- POUs/IO/Drives/SoE/Ax5000ParamSTRUCTs/P/AX5000_P_0127.TcDUT
TYPE AX5000_P_0127 :
STRUCT
	Actual_lenght:UINT;
	Max_lenght:UINT;
	Coil_unit_mass:UDINT;
	Load_mass:UDINT;
END_STRUCT
END_TYPE

// ---- POUs/IO/Drives/SoE/Ax5000ParamSTRUCTs/P/AX5000_P_0170.TcDUT
TYPE AX5000_P_0170 :
STRUCT
	Feedback_data_state:UINT;
END_STRUCT
END_TYPE

// ---- POUs/IO/Drives/SoE/Ax5000ParamSTRUCTs/P/AX5000_P_0181.TcDUT
{attribute 'pack_mode' := '1'}//Ensures 1-byte-alignmend
TYPE AX5000_P_0181 :
STRUCT
	Actual_lenght:UINT;
	Max_lenght:UINT;
	Manufacturer:UINT;
	Feedback_type:UINT;
	Feedback_type_string:STRING(29);
//	{attribute 'hide'}
	Rsvd1:ARRAY[0..4] OF UINT;
	Process_channel:ARRAY[0..11] OF UINT;
	Parameter_channel:ARRAY[0..77] OF UINT;
	Manufacturer_limits_settings:ARRAY[0..5] OF UINT;
//	{attribute 'hide'}
	Rsvd2:ARRAY[0..7] OF UINT;
END_STRUCT
END_TYPE

// ---- POUs/IO/Drives/SoE/Ax5000ParamSTRUCTs/P/AX5000_P_0198.TcDUT
{attribute 'pack_mode' := '1'}//Ensures 1-byte-alignmend
TYPE AX5000_P_0198 :
STRUCT
	Actual_lenght:UINT;
	Max_lenght:UINT;
	Feedback_instance:UINT;
	Cmd:UINT;
	Timeout:UINT;
	Byte_length:UINT;
	Addr:UDINT;
	Byte2_length:UINT;
	Error_code_as_response:UINT;
	Data: ARRAY [0..3] OF UINT;
END_STRUCT
END_TYPE

// ---- POUs/IO/Drives/SoE/Ax5000ParamSTRUCTs/P/AX5000_P_0200.TcDUT
TYPE AX5000_P_0200 :
STRUCT
	Actual_main_voltage_peak_value:UINT;
END_STRUCT
END_TYPE

// ---- POUs/IO/Drives/SoE/Ax5000ParamSTRUCTs/P/AX5000_P_0202.TcDUT
TYPE AX5000_P_0202 :
STRUCT
	Main_voltage_positive_tolerance_range:UINT;
END_STRUCT
END_TYPE

// ---- POUs/IO/Drives/SoE/Ax5000ParamSTRUCTs/P/AX5000_P_0206.TcDUT
{attribute 'pack_mode' := '1'}//Ensures 1-byte-alignmend
TYPE AX5000_P_0206 :
STRUCT
	Actual_lenght:UINT;
	Max_lenght:UINT;
	Umain_max_critical_hardware_voltage:UINT;
	Umain_min_critical_hardware_voltage:UINT;
	Umain_overvoltage_threshold:UINT;
	Umain_underervoltage_threshold:UINT;
	Umain_peak_overvoltage_threshold:UINT;
	Umain_peak_underervoltage_threshold:UINT;
	Umain_peak_lost_phase_threshold:UINT;
	Internal_brake_chopper_on_threshold:UINT;
	Internal_brake_chopper_off_threshold:UINT;
	Base_internal_brake_chopper_on_threshold:UINT;
	External_brake_chopper_on_threshold:UINT;
	External_brake_chopper_off_threshold:UINT;
	Base_external_brake_chopper_on_threshold:UINT;
	External_dc_link_connection_off_threshold:UINT;
	DCLink_volervoltage_on_threshold:UINT;
	DCLink_undervoltage_off_threshold:UINT;
	DCLink_undervoltage_warning_threshold:UINT;
	DCLink_undervoltage_error_threshold:UINT;
	DCLink_bypass_load_resistor_on_threshold:UINT;
	DCLink_bypass_load_resistor_off_threshold:UINT;
	External_Umain_rekay_off_threshold:UINT;
	External_Umain_rekay_on_threshold:UINT;
	AX5160_AX5193_Umain_peak_phase_monitoring_threshold:UINT;
//	{attribute 'hide'}
	Rsvd:ARRAY[0..6] OF UINT;

END_STRUCT
END_TYPE

// ---- POUs/IO/Drives/SoE/Ax5000ParamSTRUCTs/P/AX5000_P_0207.TcDUT
{attribute 'pack_mode' := '1'}//Ensures 1-byte-alignmend
TYPE AX5000_P_0207 :
STRUCT
	Actual_lenght:UINT;
	Max_lenght:UINT;
	Resistance:UINT;
	Continuous_Power:UINT;
	Period_time_for_duty_cycle:UINT;
	Break_resistor_protection:UINT;
	Maximum_peak_energy_by_40Percent_duty_cycle:UDINT;
	Maximum_peak_energy_by_20Percent_duty_cycle:UDINT;
	Maximum_peak_energy_by_10Percent_duty_cycle:UDINT;
	Maximum_peak_energy_by_1Percent_duty_cycle:UDINT;
	Maximum_peak_energy_by_01Percent_duty_cycle:UDINT;
	Rsvd:ARRAY[0..3] OF UDINT;

END_STRUCT
END_TYPE

// ---- POUs/IO/Drives/SoE/Ax5000ParamSTRUCTs/P/AX5000_P_0208.TcDUT
{attribute 'pack_mode' := '1'}//Ensures 1-byte-alignmend
TYPE AX5000_P_0208 :
STRUCT
	Actual_lenght:UINT;
	Max_lenght:UINT;
	Resistance:UINT;
	Continuous_Power:UINT;
	Period_time_for_duty_cycle:UINT;
	Break_resistor_protection:UINT;
	Maximum_peak_energy_by_40Percent_duty_cycle:UDINT;
	Maximum_peak_energy_by_20Percent_duty_cycle:UDINT;
	Maximum_peak_energy_by_10Percent_duty_cycle:UDINT;
	Maximum_peak_energy_by_1Percent_duty_cycle:UDINT;
	Maximum_peak_energy_by_01Percent_duty_cycle:UDINT;
	Rsvd:ARRAY[0..3] OF UDINT;

END_STRUCT
END_TYPE

// ---- POUs/IO/Drives/SoE/Ax5000ParamSTRUCTs/P/AX5000_P_0209.TcDUT
TYPE AX5000_P_0209 :
STRUCT
	Internal_brak_resistor_actual_continouse_power:UINT;
END_STRUCT
END_TYPE

// ---- POUs/IO/Drives/SoE/Ax5000ParamSTRUCTs/P/AX5000_P_0211.TcDUT
TYPE AX5000_P_0211 :
STRUCT
	Warning_level_Actual_cont_power_internal_brake_resistor:UINT;
END_STRUCT
END_TYPE

// ---- POUs/IO/Drives/SoE/Ax5000ParamSTRUCTs/P/AX5000_P_0217.TcDUT
TYPE AX5000_P_0217 :
STRUCT
	Actual_main_voltage:UINT;
END_STRUCT
END_TYPE

// ---- POUs/IO/Drives/SoE/Ax5000ParamSTRUCTs/P/AX5000_P_0254.TcDUT
TYPE AX5000_P_0254 :
STRUCT
	Probe_1_time_negative_edge:UDINT;
END_STRUCT
END_TYPE

// ---- POUs/IO/Drives/SoE/Ax5000ParamSTRUCTs/P/AX5000_P_0302.TcDUT
TYPE AX5000_P_0302 :
STRUCT
	Display_value_line_1:UINT;
END_STRUCT
END_TYPE

// ---- POUs/IO/Drives/SoE/Ax5000ParamSTRUCTs/P/AX5000_P_0352.TcDUT
TYPE AX5000_P_0352 :
STRUCT
	Drive_halt_jerk_bipolar:UDINT;
END_STRUCT
END_TYPE

// ---- POUs/IO/Drives/SoE/Ax5000ParamSTRUCTs/P/AX5000_P_0354.TcDUT
TYPE AX5000_P_0354 :
STRUCT
	Standstill_window_monitoring_time:UINT;
END_STRUCT
END_TYPE

// ---- POUs/IO/Drives/SoE/Ax5000ParamSTRUCTs/P/AX5000_P_0464.TcDUT
{attribute 'pack_mode' := '1'}
TYPE AX5000_P_0464 :
STRUCT
	Actual_lenght:UINT;
	Max_lenght:UINT;
	Mode:UINT;
	Adaptive_gain:UINT;
	Min_bandswitch:UINT;
	Max_bandswitch:UINT;
	Correction_factor_Iq_to_Acc:UINT;
	Damping:UINT;
	Starting_current_command:UINT;
	Rsvd:UINT;
	Threshold_speed1:UDINT;
	Threshold_speed2:UDINT;
//	{attribute 'hide'}
	Rsvd2:UDINT;
END_STRUCT
END_TYPE

// ---- POUs/IO/Drives/SoE/Ax5000ParamSTRUCTs/P/AX5000_P_0505.TcDUT
TYPE AX5000_P_0505 :
STRUCT
	Velocity_controller_output:UINT;
END_STRUCT
END_TYPE

// ---- POUs/IO/Drives/SoE/Ax5000ParamSTRUCTs/P/AX5000_P_0514.TcDUT
{attribute 'pack_mode' := '1'}
TYPE AX5000_P_0514 :
STRUCT
	Actual_lenght:UINT;
	Max_lenght:UINT;
	Mode:UINT;
//	{attribute 'hide'}
	Rsvd1:UINT;
	Bandswitch:UINT;
	Correction_factor_Iq_to_acc:UINT;
	Damping:UINT;
//	{attribute 'hide'}
	Rsvd2:UINT;
END_STRUCT
END_TYPE

// ---- POUs/IO/Drives/SoE/Ax5000ParamSTRUCTs/P/AX5000_P_0516.TcDUT
{attribute 'pack_mode' := '1'}
TYPE AX5000_P_0516 :
STRUCT
	Actual_lenght:UINT;
	Max_lenght:UINT;
	ST_CONV_Version:UINT;
	Rsvd1:UINT;
	Filter_type:UINT;
//	{attribute 'hide'}
	Rsvd2:UINT;
	Low_pass_frequency:UDINT;
	Low_pass_damping:UDINT;
	High_pass_frequency:UDINT;
	High_pass_damping:UDINT;
//	{attribute 'hide'}
	Rsvd3:UDINT;
//	{attribute 'hide'}
	Rsvd4:UDINT;
	QMath_factor:UINT;
//	{attribute 'hide'}
	Rsvd5:UINT;
	b0:UDINT;
	b1:UDINT;
	b2:UDINT;
	a1:UDINT;
	a2:UDINT;
//	{attribute 'hide'}
	Rsvd6:UDINT;
	Rsvd7:UDINT;
END_STRUCT
END_TYPE

// ---- POUs/IO/Drives/SoE/Ax5000ParamSTRUCTs/P/AX5000_P_0557.TcDUT
TYPE AX5000_P_0557 :
STRUCT
	Acceleration_feedforward_filter_timeconstant:UINT;
END_STRUCT
END_TYPE

// ---- POUs/IO/Drives/SoE/Ax5000ParamSTRUCTs/P/AX5000_P_0811.TcDUT
TYPE AX5000_P_0811 :
STRUCT
	Customer_specific_functionality_status:UDINT;
END_STRUCT
END_TYPE

// ---- POUs/IO/Drives/SoE/Ax5000ParamSTRUCTs/P/AX5000_P_0900.TcDUT
TYPE AX5000_P_0900 :
STRUCT
	Actual_lenght:UINT;
	Max_lenght:UINT;
(*Control Pcb*)
	Safety_test_status:UINT;
//	{attribute 'hide'}
	Rsvd1:UINT;
	Channel0_offset:INT;
	Channel0_gain:UINT;
	Channel1_offset:INT;
	Channel1_gain:UINT;
	Channel2_offset:INT;
	Channel2_gain:UINT;
	Channel3_offset:INT;
	Channel3_gain:UINT;
	Channel4_offset:INT;
	Channel4_gain:UINT;
	Channel5_offset:INT;
	Channel5_gain:UINT;
	Channel6_offset:INT;
	Channel6_gain:UINT;
	Channel7_offset:INT;
	Channel7_gain:UINT;
	Channel8_offset:INT;
	Channel8_gain:UINT;
	Channel9_offset:INT;
	Channel9_gain:UINT;
//	{attribute 'hide'}
	Rsvd2:ARRAY[0..6] OF UINT;
	Checksum:UINT;

(*Power Pcb*)
	(*Ch A*)
	ChA_Calibration_type:UINT;
	ChA_V_Offset:INT;
	ChA_W_Offset:INT;
	ChA_V_resistor_value1:UINT;
	ChA_W_resistor_value1:UINT;
	ChA_V_resistor_value2:UINT;
	ChA_W_resistor_value2:UINT;
	ChA_V_resistor_value3:UINT;
	ChA_W_resistor_value3:UINT;
	ChA_V_resistor_value4:UINT;
	ChA_W_resistor_value4:UINT;
	ChA_V_current_value1:UINT;
	ChA_W_current_value1:UINT;
	ChA_V_current_value2:UINT;
	ChA_W_current_value2:UINT;
	ChA_V_current_value3:UINT;
	ChA_W_current_value3:UINT;
	ChA_V_current_value4:UINT;
	ChA_W_current_value4:UINT;
	(*Ch B*)
	ChB_Calibration_type:UINT;
	ChB_V_Offset:INT;
	ChB_W_Offset:INT;
	ChB_V_resistor_value1:UINT;
	ChB_W_resistor_value1:UINT;
	ChB_V_resistor_value2:UINT;
	ChB_W_resistor_value2:UINT;
	ChB_V_resistor_value3:UINT;
	ChB_W_resistor_value3:UINT;
	ChB_V_resistor_value4:UINT;
	ChB_W_resistor_value4:UINT;
	ChB_V_current_value1:UINT;
	ChB_W_current_value1:UINT;
	ChB_V_current_value2:UINT;
	ChB_W_current_value2:UINT;
	ChB_V_current_value3:UINT;
	ChB_W_current_value3:UINT;
	ChB_V_current_value4:UINT;
	ChB_W_current_value4:UINT;
//	{attribute 'hide'}
	Rsvd3:UINT;
	Checksum2:UINT;

(*Driver Pcb*)
	Safety_test_status2:UINT;
	Calibration_type2:UINT;
//	{attribute 'hide'}
	Rsvd4:UINT;
	Udclink_offset:UINT;
	Udclink_gain:UINT;
	Udclink_offset1:UINT;
	Udclink_gain1:UINT;
	Udclink_offset2:UINT;
	Udclink_gain2:UINT;
	Udclink_offset3:UINT;
	Udclink_gain3:UINT;
//	{attribute 'hide'}
	Rsvd5:ARRAY[0..17] OF UINT;
	Checksum3:UINT;

(*Front Pcb*)
	Vendor:UDINT;
	Product_code:UDINT;
	Revision_No:UDINT;
	Serial_No:UDINT;
	Year:USINT;
	Week:USINT;
	Fan_profiltype_internalbrakeresistor_rsvd:UINT;		(*jeweils 4 Bit*)
	Hardware_device_id_2:UINT;
	Hardware_device_id_3:UINT;
	Hardware_device_id_4:UINT;
//	{attribute 'hide'}
	Rsvd6:ARRAY[0..2] OF UINT;
	Customized_id:UINT;
	ModificationId:UINT;
//	{attribute 'hide'}
	Rsvd7:ARRAY[0..3] OF UINT;
	Free_switch_code1:UINT;
	Free_switch_code2:UINT;
//	{attribute 'hide'}
	Rsvd8:ARRAY[0..3] OF UINT;
	ST_CONV_Version:UINT;
//	{attribute 'hide'}
	Rsvd9:UINT;
	(*ChA*)
	ChA_Sin_offset:DINT;
	ChA_Cos_offset:DINT;
	ChA_Sin_gain:UDINT;
	ChA_Cos_gain:UDINT;
	ChA_Excitation_voltage_Gain:UINT;
	ChA_rsvd10:ARRAY[0..2] OF UINT;
	(*ChB*)
	ChB_Sin_offset:DINT;
	ChB_Cos_offset:DINT;
	ChB_Sin_gain:UDINT;
	ChB_Cos_gain:UDINT;
	ChB_Excitation_voltage_Gain:UINT;
	ChB_rsvd11:ARRAY[0..2] OF UINT;
//{attribute 'hide'}
	Rsvd12:ARRAY[0..24] OF UINT;
	Checksum4:UINT;

(*Option Pcb*)
	Vendor2:UDINT;
	Product_code2:UDINT;
	Revision_No2:UDINT;
	Serial_No2:UDINT;
	Year2:USINT;
	Week2:USINT;
	Fan_profiltype_internalbrakeresistor_rsvd2:UINT;		(*jeweils 4 Bit*)
	Hardware_device_id_22:UINT;
	Hardware_device_id_32:UINT;
	Hardware_device_id_42:UINT;
//	{attribute 'hide'}
	Rsvd13:ARRAY[0..2] OF UINT;
	Customized_id2:UINT;
	ModificationId2:UINT;
//	{attribute 'hide'}
	Rsvd14:ARRAY[0..3] OF UINT;
	Free_switch_code12:UINT;
	Free_switch_code22:UINT;
//	{attribute 'hide'}
	Rsvd15:ARRAY[0..3] OF UINT;
	Version2:UINT;
//	{attribute 'hide'}
	Rsvd16:UINT;
	(*ChA*)
	ChA_Sin_offset2:DINT;
	ChA_Cos_offset2:DINT;
	ChA_Sin_gain2:UDINT;
	ChA_Cos_gain2:UDINT;
	ChA_Excitation_voltage_Gai2n:UINT;
	ChA_rsvd17:ARRAY[0..2] OF UINT;
	(*ChB*)
	ChB_Sin_offset2:DINT;
	ChB_Cos_offse2t:DINT;
	ChB_Sin_gain2:UDINT;
	ChB_Cos_gain2:UDINT;
	ChB_Excitation_voltage_Gai2n:UINT;
	ChB_rsvd18:ARRAY[0..2] OF UINT;
//{attribute 'hide'}
	Rsvd19:ARRAY[0..24] OF UINT;
	Checksum5:UINT;

(*Safety Pcb*)
//{attribute 'hide'}
	Rsvd20:ARRAY[0..8] OF UINT;
	Checksum6:UINT;

	Control_Pcb_data_valid:UINT;
	Power_Pcb_data_valid:UINT;
	Driver_Pcb_data_valid:UINT;
	Front_Pcb_data_valid:UINT;
	Option_Pcb_data_valid:UINT;
	Safety_Pcb_data_valid:UINT;

END_STRUCT
END_TYPE

// ---- POUs/IO/Drives/SoE/Ax5000ParamSTRUCTs/P/AX5000_P_1009.TcDUT
TYPE AX5000_P_1009 :
STRUCT
	Addr:UINT;
	Source:UINT;
END_STRUCT
END_TYPE

// ---- POUs/IO/Drives/SoE/Ax5000ParamSTRUCTs/P/AX5000_P_1010.TcDUT
TYPE AX5000_P_1010 :
STRUCT
	Feedback_debug_pointer_2_vtype:UINT;
END_STRUCT
END_TYPE

// ---- POUs/IO/Drives/SoE/Ax5000ParamSTRUCTs/S/AX5000_S_0016.TcDUT
TYPE AX5000_S_0016 :
STRUCT
	Actual_lenght:UINT;
	Max_lenght:UINT;
	Configuration_list_of_AT:ARRAY[0..23] OF UINT;
END_STRUCT
END_TYPE

// ---- POUs/IO/Drives/SoE/Ax5000ParamSTRUCTs/S/AX5000_S_0024.TcDUT
TYPE AX5000_S_0024 :
STRUCT
	Actual_lenght:UINT;
	Max_lenght:UINT;
	Configuration_list_of_MDT:ARRAY[0..11] OF UINT;
END_STRUCT
END_TYPE

// ---- POUs/IO/Drives/SoE/Ax5000ParamSTRUCTs/S/AX5000_S_0029.TcDUT
TYPE AX5000_S_0029 :
STRUCT
	MDT_error_counter:UINT;
END_STRUCT
END_TYPE

// ---- POUs/IO/Drives/SoE/Ax5000ParamSTRUCTs/S/AX5000_S_0032.TcDUT
TYPE AX5000_S_0032 :
STRUCT
	Primary_operation_mode:E_AX5000_S_0032_OperationMode;
END_STRUCT
END_TYPE

// ---- POUs/IO/Drives/SoE/Ax5000ParamSTRUCTs/S/AX5000_S_0035.TcDUT
TYPE AX5000_S_0035 :
STRUCT
	Secondary_operation_mode3:UINT;
END_STRUCT
END_TYPE

// ---- POUs/IO/Drives/SoE/Ax5000ParamSTRUCTs/S/AX5000_S_0036.TcDUT
TYPE AX5000_S_0036 :
STRUCT
	Velocity_command_value:DINT;
END_STRUCT
END_TYPE

// ---- POUs/IO/Drives/SoE/Ax5000ParamSTRUCTs/S/AX5000_S_0055.TcDUT
TYPE AX5000_S_0055 :
STRUCT
	Position_polatity_parameter:UINT;
END_STRUCT
END_TYPE

// ---- POUs/IO/Drives/SoE/Ax5000ParamSTRUCTs/S/AX5000_S_0082.TcDUT
TYPE AX5000_S_0082 :
STRUCT
	Positiv_Torque_command_value:UINT;
END_STRUCT
END_TYPE

// ---- POUs/IO/Drives/SoE/Ax5000ParamSTRUCTs/S/AX5000_S_0083.TcDUT
TYPE AX5000_S_0083 :
STRUCT
	Negative_Torque_command_value:UINT;
END_STRUCT
END_TYPE

// ---- POUs/IO/Drives/SoE/Ax5000ParamSTRUCTs/S/AX5000_S_0112.TcDUT
TYPE AX5000_S_0112 :
STRUCT
	Amplifier_rated_current:UDINT;
END_STRUCT
END_TYPE

// ---- POUs/IO/Drives/SoE/Ax5000ParamSTRUCTs/S/AX5000_S_0295.TcDUT
TYPE AX5000_S_0295 :
STRUCT
	Drive_enable_delay_time:UINT;
END_STRUCT
END_TYPE

// ---- POUs/IO/Drives/SoE/Ax5000ParamSTRUCTs/S/AX5000_S_0348.TcDUT
TYPE AX5000_S_0348 :
STRUCT
	Acceleration_feed_forword_gain:UINT;
END_STRUCT
END_TYPE

// ---- POUs/IO/_ItfActuators/I_ActuatorPosNeg.TcIO
INTERFACE I_ActuatorPosNeg EXTENDS I_ActuatorBase

{attribute 'monitoring' := 'call'}
PROPERTY public negativeOk : BOOL
GET
END_GET
END_PROPERTY

METHOD PUBLIC negativeOn : BOOL
VAR_INPUT
END_VAR
END_METHOD

{attribute 'monitoring' := 'call'}
PROPERTY public positiveOk : BOOL
GET
END_GET
END_PROPERTY

METHOD PUBLIC positiveOn : BOOL
VAR_INPUT
END_VAR
END_METHOD

END_INTERFACE

// ---- POUs/IO/_ItfActuators/I_ActuatorUpDown.TcIO
INTERFACE I_ActuatorUpDown EXTENDS I_ActuatorBase

{attribute 'monitoring' := 'call'}
PROPERTY public downOk : BOOL
GET
END_GET
END_PROPERTY

METHOD public moveDown : BOOL
VAR_INPUT
END_VAR
END_METHOD

METHOD public moveUp : BOOL
VAR_INPUT
END_VAR
END_METHOD

{attribute 'monitoring' := 'call'}
PROPERTY public upOK : BOOL
GET
END_GET
END_PROPERTY

END_INTERFACE

// ---- POUs/Logging/I_LogbookSubscriber.TcIO
INTERFACE I_LogbookSubscriber Extends __System.IQueryInterface

METHOD addNewMessage : BOOL
VAR_IN_OUT
	data										:	LogbookData;
END_VAR
END_METHOD

{attribute 'monitoring' := 'call'}
PROPERTY PUBLIC isBusy : BOOL
GET
END_GET
END_PROPERTY

END_INTERFACE

// ---- POUs/Connectivity/ADS/AdsDataExchange.TcPOU
//"DataExchange" enables a ADS communication by symbol name between two TwinCAT runtime system
//based on Tc2_System
{attribute 'no_check'}
FUNCTION_BLOCK AdsDataExchange
VAR_OUTPUT CONSTANT
	MODE_FETCH_CONTINOUS									:	INT := 0;
	MODE_FETCH_BY_EVENT										:	INT := 1;
	MODE_SEND_CONTINOUS										:	INT := 2;
	MODE_SEND_BY_EVENT										:	INT := 3;
END_VAR
VAR_IN_OUT
END_VAR
VAR_INPUT
	Enable													:	BOOL := FALSE;	// FB will be processed as long as enable is TRUE 
	Transmit												:	BOOL := FALSE;	// TRUE or a rising edge starts the data exchange - depends on requested mode 
	Mode													:	INT (MODE_FETCH_CONTINOUS..MODE_SEND_BY_EVENT ) := MODE_SEND_BY_EVENT; //requested modes
	NetId													:	T_AmsNetId := ''; // Target AMS-NetID or '' for local-target
	Port													:	T_AmsPort := 851; 	// ADS-Communication-Port (PLC Runtime Port)
	DestSymbol												:	STRING;			//Desination symbol name to fetch or send - depends on requested mode
	pData													:	PVOID := 0;		//Pointer of data to send or target to fetch data - depends on requested mode 
	cbData													:	UDINT := 0;		//Data size of data to send or target to fetch data - depends on requested mode 
	Timeout													:	TIME := DEFAULT_ADS_TIMEOUT;// timeout for ADS request
END_VAR
VAR_OUTPUT
	hSymbol													:	UDINT;	//Symbol handle
	Ready													:	BOOL;	//ADS Route initialized successfully and ready to send/fetch											
	Active													:	BOOL;	//communication data exchange is in process (transmit triggered=
	Busy													:	BOOL; 	//Busy is TRUE at the rising edge of Enable and stays TRUE as long as the FB is performing any action. 
	Error													:	BOOL;	//Rising edge of Error informs that an error occurred during the execution of the Function Block  
{attribute 'displaymode':='hex'}
	ErrorID													:	UDINT; 	//Error identification - see ADS return codes at Beckhoff infosys for further information 
END_VAR
VAR
(* local variables *****************************************************)
	state													: 	INT := 0;
	MemErrorId												:	UDINT := 0;
	
(* trigger **********************************************************)
	FT_Enable												:	F_TRIG;
	RT_Transmit												:	R_TRIG;

(* timer ************************************************************)

(* finstances ***************************************************************)
	AdsRdWr_CreateVar_H										:	ADSRDWRT;
	FetchVal_ReqVar											:	ADSREAD;
	SendVal_ReqVar											:	ADSWRITE;
	ReleaseSymHandle										:	ADSWRITE;
END_VAR

FT_Enable(CLK 	:= Enable); // necessary for handle release 
RT_Transmit(CLK := Transmit AND Ready); // necessary for event mode

(* Sequence ********************************************************************************)
IF Enable THEN
	CASE state OF
	0: //Start creating symbol handle
		//Init fbs		
		AdsRdWr_CreateVar_H(WRTRD := FALSE);
		FetchVal_ReqVar(READ := FALSE);
		SendVal_ReqVar(WRITE := FALSE);
		ReleaseSymHandle(WRITE := FALSE);
		
		Busy 												:= TRUE;
		
		IF NOT AdsRdWr_CreateVar_H.BUSY AND NOT FetchVal_ReqVar.BUSY
			AND NOT SendVal_ReqVar.BUSY AND NOT ReleaseSymHandle.BUSY
		THEN
			AdsRdWr_CreateVar_H(NETID := NETID, PORT := PORT,
								IDXGRP := ADSIGRP_SYM_HNDBYNAME, IDXOFFS := 0,
								WRITELEN := SIZEOF(DestSymbol),// max. no. of chars req. variable
								READLEN := SIZEOF(hSymbol),
								SRCADDR := ADR(DestSymbol)	, DESTADDR := ADR(hSymbol), WRTRD := TRUE, TMOUT := Timeout);
			state											:= state + 1;						
		END_IF


	1://Wait for symbol handle 
		AdsRdWr_CreateVar_H(NETID := NETID, PORT := PORT,
							IDXGRP := ADSIGRP_SYM_HNDBYNAME, IDXOFFS := 0,
							WRITELEN := SIZEOF(DestSymbol),// max. no. of chars req. variable
							READLEN := SIZEOF(hSymbol),
							SRCADDR := ADR(DestSymbol)	, DESTADDR := ADR(hSymbol), WRTRD := TRUE, TMOUT := Timeout);	
		IF NOT AdsRdWr_CreateVar_H.BUSY
		THEN
			IF AdsRdWr_CreateVar_H.ERR
			THEN
				Busy										:= FALSE;
				Error										:= TRUE;
				ErrorId										:= AdsRdWr_CreateVar_H.ERRID;
				state										:= state * -1;
			ELSE
				Ready										:= TRUE;
				state										:= state + 1;
			END_IF
			AdsRdWr_CreateVar_H(WRTRD := FALSE);
		END_IF
		
	2: //Start fetch or send data 
		IF RT_Transmit.Q AND Mode = MODE_FETCH_BY_EVENT 
			OR Mode = MODE_FETCH_CONTINOUS
		THEN	
		 	FetchVal_ReqVar(	
				NETID 	:= NETID, 
				PORT 	:= PORT, 
				TMOUT 	:= Timeout,
				IDXGRP 	:= ADSIGRP_SYM_VALBYHND, 
				IDXOFFS := hSymbol, 	
				LEN 	:= cbData, 	
				DESTADDR:= pData,
				READ 	:= TRUE);
			Active											:= TRUE;
			state											:= state + 1;
		ELSIF RT_Transmit.Q AND Mode = MODE_SEND_BY_EVENT 
			OR Mode = MODE_SEND_CONTINOUS
		THEN 
			SendVal_ReqVar( 
				NETID 	:= NETID, 
				PORT 	:= PORT, 
				TMOUT 	:= Timeout,
				IDXGRP 	:= ADSIGRP_SYM_VALBYHND, 
				IDXOFFS	:= hSymbol, 
				SRCADDR := pData,
				LEN		:= cbData,  
				WRITE 	:= TRUE);		
			Active											:= TRUE;
			state											:= state + 1;
		END_IF
		
	3: //Wait for send/fetch done 
		IF FetchVal_ReqVar.READ
		THEN
		 	FetchVal_ReqVar(LEN 	:= cbData, DESTADDR:= pData, READ 	:= TRUE);		
			IF NOT FetchVal_ReqVar.BUSY
			THEN
				Active										:= FALSE;
				IF FetchVal_ReqVar.ERR
				THEN
					Busy									:= FALSE;
					Error									:= TRUE;
					ErrorId									:= FetchVal_ReqVar.ERRID;
					state									:= state * -1;					
				ELSE
					Ready									:= TRUE;
					state 									:= state - 1;
				END_IF
				FetchVal_ReqVar(READ 	:= FALSE);
			END_IF
		
		ELSE
			SendVal_ReqVar( SRCADDR := pData,LEN := cbData,  WRITE 	:= TRUE);	
			IF NOT SendVal_ReqVar.BUSY
			THEN		
				Active										:= FALSE;
				IF SendVal_ReqVar.ERR
				THEN
					Busy									:= FALSE;
					Error									:= TRUE;
					ErrorId									:= SendVal_ReqVar.ERRID;
					state									:= state * -1;					
				ELSE
					Ready									:= TRUE;
					state 									:= state - 1;
				END_IF
				SendVal_ReqVar(WRITE 	:= FALSE);		
			END_IF
		END_IF
	ELSE //Error - wait for enable = FALSE	
		MemErrorId											:= ErrorId;
 	END_CASE
ELSE //Enable = FALSE	
	Active													:= FALSE;
	Ready													:= FALSE;
	IF FT_Enable.Q 
	THEN  
		ReleaseSymHandle(WRITE:= FALSE);
		ReleaseSymHandle(NETID := NETID, 
						PORT 	:= PORT, 
						TMOUT 	:= Timeout,
						IDXGRP 	:= ADSIGRP_SYM_RELEASEHND, 
						IDXOFFS := hSymbol, 
						LEN 	:= 0, 
						WRITE 	:= hSymbol <> 0);
	ELSE
		ReleaseSymHandle();
		IF NOT ReleaseSymHandle.BUSY
		THEN
			ReleaseSymHandle(Write := FALSE);
			hSymbol											:= 0;
			Error 											:= FALSE;		
			ErrorID 										:= 0;
			Busy 											:= FALSE;
			State	 										:= 0;				
		END_IF
	END_IF

END_IF
	
(*********************************************************************************************************)

END_FUNCTION_BLOCK

// ---- POUs/Connectivity/Ipv4Addr_TO_UDINT.TcPOU
//Converts an IPv4 address string to a hex coded UDINT
	{attribute 'displaymode':='hex'}
FUNCTION Ipv4Addr_TO_UDINT : UDINT
VAR_INPUT
	IPv4Addr				:	T_IPv4Addr; //String
END_VAR
VAR
	Bytes 					: 	T_IPv4AddrArr; //IPv4 address as an array 0..3 of Byte
END_VAR

Bytes						:= F_ScanIPv4AddrIds(IPv4Addr);
MEMCPY(ADR(Ipv4Addr_TO_UDINT),ADR(Bytes[3]),1);
MEMCPY(ADR(Ipv4Addr_TO_UDINT)+1,ADR(Bytes[2]),1);
MEMCPY(ADR(Ipv4Addr_TO_UDINT)+2,ADR(Bytes[1]),1);
MEMCPY(ADR(Ipv4Addr_TO_UDINT)+3,ADR(Bytes[0]),1);

END_FUNCTION

// ---- POUs/Connectivity/TF625x-Modbus/Master/TF6250-ModbusTcpServer/UDP/ModbusUdpMaster.TcPOU
{attribute 'no_check'}
// ModBus comunication master to multible slaves useing UDP protocol
// based on TF6250 - required lib: Tc2_ModbusTCP
FUNCTION_BLOCK ModbusUdpMaster
VAR CONSTANT
	MIN_SLAVE												:	INT := 1;
	MAX_SLAVE												:	INT := PARAM.MODBUS_MAX_SLAVES_OF_MASTER;
END_VAR
VAR_INPUT
	Enable													:	BOOL ; 		// FB will be processed as long as enable is TRUE 
	ResetTrig												:	BOOL ;		// The function block will be reset with a rising edge 
	SlaveCom												:	ARRAY[MIN_SLAVE..MAX_SLAVE] OF POINTER TO ModbusSlaveCom;
	Timestamp												:	DT;
END_VAR         	
VAR_OUTPUT      	
	Error													:	BOOL;		// Rising edge of Error informs that an error occurred during the execution of the Function Block 
{attribute 'displaymode':='hex'}
	ErrorID													:	UDINT;		// Error identification - see ADS return codes at Beckhoff infosys for further information 
	ErrorText												:	STRING;
END_VAR
VAR
(* memory **************************************************)
	state 													:	INT := 0;
	JobNo													:	INT := 0;
	SlaveNo													:	INT := 0;
(* trigger *************************************************)

(* timer ***************************************************)

(* blocks **************************************************)
	ReadCoils												:	FB_MBUdpReadCoils := (tTimeout		:= DEFAULT_ADS_TIMEOUT);		// Fnc 1
	ReadInputs												:	FB_MBUdpReadInputs := (tTimeout		:= DEFAULT_ADS_TIMEOUT);		// Fnc 2
	ReadRegs												:	FB_MBUdpReadRegs := (tTimeout		:= DEFAULT_ADS_TIMEOUT);		// Fnc 3
	ReadInputRegs											:	FB_MBUdpReadInputRegs := (tTimeout	:= DEFAULT_ADS_TIMEOUT);	// Fnc 4
	WriteSingleCoil											:	FB_MBUdpWriteSingleCoil := (tTimeout:= DEFAULT_ADS_TIMEOUT);// Fnc 5
	WriteSingleReg											:	FB_MBUdpWriteSingleReg := (tTimeout	:= DEFAULT_ADS_TIMEOUT);	// Fnc 6
	Diagnose												:	FB_MBUdpDiagnose := (tTimeout		:= DEFAULT_ADS_TIMEOUT);		// Fnc 8
	WriteCoils												:	FB_MBUdpWriteCoils := (tTimeout		:= DEFAULT_ADS_TIMEOUT);		// Fnc 15
	WriteRegs												:	FB_MBUdpWriteRegs := (tTimeout		:= DEFAULT_ADS_TIMEOUT);		// Fnc 16
	ReadWriteRegs											:	FB_MBUdpReadWriteRegs := (tTimeout	:= DEFAULT_ADS_TIMEOUT); 	// Fnc 23	use read and write job instead
(* internal used variables *********************************)
	i,j,k													:	INT :=0;
END_VAR


	CASE state OF
	0:	(* Idle *)
		IF Enable 
		THEN
			k 												:=	0;
			JobNo  :=  SlaveNo								:=	1;
			state 											:=	10;
		END_IF

	10: 
		IF GetNextSlave() 
		THEN (* find Slave *)
			k 												:= 0;
			IF GetNextJob() 
			THEN (* find JobNo *)
				SlaveCom[SlaveNo]^.currentJobIdx 			:= JobNo;
				SlaveCom[SlaveNo]^.writeJobRequested 		:= SlaveCom[SlaveNo]^.Jobs[JobNo].FunctionCode >= 5;
				State 										:= SEL(SlaveCom[SlaveNo]^.writeJobRequested, 20, 15);
			END_IF
		ELSE
			state 											:=	0;
		END_IF
	
	15: (* wait for valid write date *)
		IF NOT SlaveCom[SlaveNo]^.writeJobRequested
		THEN
			SlaveCom[SlaveNo]^.Jobs[JobNo].Valid 			:= FALSE;
			state 											:= 20;
		END_IF

	20: (* start job *)	
		IF NOT StartJob(FALSE) // Busy
		THEN						
			state 											:= 30;
		END_IF

	30: (* wait for com cycle *)
		IF NOT StartJob(TRUE) THEN // Busy
			IF Error 
			THEN
				ErrorText									:= CONCAT('Error at SlaveNo: ',	CONCAT(INT_TO_STRING(SlaveNo), CONCAT(', JobNo: ', INT_TO_STRING(JobNo))));
				SlaveCom[SlaveNo]^.countBad 				:= SlaveCom[SlaveNo]^.countBad +1;
				state 										:= 98; 
			ELSE
				SlaveCom[SlaveNo]^.countGood 				:= SlaveCom[SlaveNo]^.countGood +1;
				SlaveCom[SlaveNo]^.Jobs[JobNo].Valid 		:= TRUE;
				SlaveCom[SlaveNo]^.Jobs[JobNo].TimeStamp 	:= Timestamp;
				JobNo 										:= JobNo + 1;
				state 										:= 10;	(* next job *)
			END_IF
			StartJob(FALSE);
		END_IF

	98: (* wait for quit *)
		IF ResetTrig THEN
			reset();
		END_IF

	END_CASE

METHOD PRIVATE getNextJob : Bool //Return value = TRUE if execution finished
VAR_INPUT
END_VAR
	
	WHILE SlaveCom[SlaveNo]^.Jobs[JobNo].FunctionCode = 0 DO
		JobNo 											:= JobNo + 1;
		IF JobNo > SlaveCom[SlaveNo]^.MAX_SLAVE_JOB THEN
			JobNo 										:= SlaveCom[SlaveNo]^.MIN_SLAVE_JOB;
			SlaveNo 									:= SlaveNo + 1;
			GetNextJob									:= FALSE;
			RETURN;
		END_IF
	END_WHILE
	GetNextJob											:= TRUE;
END_METHOD

METHOD PRIVATE getNextSlave : Bool //Return value = TRUE if execution finished
VAR_INPUT
END_VAR
	WHILE SlaveCom[SlaveNo] = 0 or_else not SlaveCom[SlaveNo]^.Enable DO
		SlaveNo 										:= SlaveNo + 1;
		IF SlaveNo > MAX_SLAVE 
		THEN
			k 											:= k + 1;
			SlaveNo 									:= MIN_SLAVE;
		ELSIF k = 2 
		THEN
			k 											:= 0;
			GetNextSlave								:= FALSE;
			RETURN;
		END_IF	
	END_WHILE
	GetNextSlave										:= TRUE;
END_METHOD

METHOD PUBLIC reset : booL //Return value = TRUE if execution finished
VAR_INPUT
END_VAR
IF State = 98 
THEN
	Error													:= FALSE;
	ErrorID													:= 0;
	ErrorText												:= '';
	state													:= 0;
END_IF	
reset														:= TRUE;
END_METHOD

METHOD PRIVATE startJob : BOOL //Return value = TRUE if busy - TRUE as long as the job is busy
VAR_INPUT
	Execute							: BOOL;
END_VAR
	IF 	SlaveCom[SlaveNo]^.Jobs[JobNo].FunctionCode = 1 THEN
		ReadCoils(
			sIPAddr			:= SlaveCom[SlaveNo]^.ipAddr, 
			nTCPPort		:= TO_UINT(SlaveCom[SlaveNo]^.Port), 
			nUnitID			:= SlaveCom[SlaveNo]^.Address, 
			nQuantity		:= SlaveCom[SlaveNo]^.jobs[JobNo].Quantity, 
			nMBAddr			:= SlaveCom[SlaveNo]^.jobs[JobNo].startAddress, 
			cbLength		:= SlaveCom[SlaveNo]^.jobs[JobNo].Quantity, 
			pDestAddr		:= ADR(SlaveCom[SlaveNo]^.Data), 
			bExecute		:= Execute, 
			tTimeout		:= , 
			bBusy			=> StartJob, 
			bError			=> Error, 
			nErrId			=> ErrorID);
		
	ELSIF 	SlaveCom[SlaveNo]^.Jobs[JobNo].FunctionCode = 2 THEN
		ReadInputs(
			sIPAddr			:= SlaveCom[SlaveNo]^.ipAddr, 
			nTCPPort		:= TO_UINT(SlaveCom[SlaveNo]^.Port), 
			nUnitID			:= SlaveCom[SlaveNo]^.Address, 
			nQuantity		:= SlaveCom[SlaveNo]^.jobs[JobNo].Quantity, 
			nMBAddr			:= SlaveCom[SlaveNo]^.jobs[JobNo].startAddress, 
			cbLength		:= SlaveCom[SlaveNo]^.jobs[JobNo].Quantity, 
			pDestAddr		:= ADR(SlaveCom[SlaveNo]^.Data), 
			bExecute		:= Execute, 
			tTimeout		:= , 
			bBusy			=> StartJob, 
			bError			=> Error, 
			nErrId			=> ErrorID);
			
	ELSIF 	SlaveCom[SlaveNo]^.Jobs[JobNo].FunctionCode = 3 THEN
		ReadRegs(
			sIPAddr			:= SlaveCom[SlaveNo]^.ipAddr, 
			nTCPPort		:= TO_UINT(SlaveCom[SlaveNo]^.Port), 
			nUnitID			:= SlaveCom[SlaveNo]^.Address, 
			nQuantity		:= SlaveCom[SlaveNo]^.jobs[JobNo].Quantity, 
			nMBAddr			:= SlaveCom[SlaveNo]^.jobs[JobNo].startAddress, 
			cbLength		:= SlaveCom[SlaveNo]^.jobs[JobNo].Quantity * 2, 
			pDestAddr		:= ADR(SlaveCom[SlaveNo]^.Data), 
			bExecute		:= Execute, 
			tTimeout		:= DEFAULT_ADS_TIMEOUT, 
			bBusy			=> StartJob, 
			bError			=> Error, 
			nErrId			=> ErrorID);
	
	ELSIF 	SlaveCom[SlaveNo]^.Jobs[JobNo].FunctionCode = 4 THEN
		ReadInputRegs(
			sIPAddr			:= SlaveCom[SlaveNo]^.ipAddr, 
			nTCPPort		:= TO_UINT(SlaveCom[SlaveNo]^.Port), 
			nUnitID			:= SlaveCom[SlaveNo]^.Address, 
			nQuantity		:= SlaveCom[SlaveNo]^.jobs[JobNo].Quantity, 
			nMBAddr			:= SlaveCom[SlaveNo]^.jobs[JobNo].startAddress, 
			cbLength		:= SlaveCom[SlaveNo]^.jobs[JobNo].Quantity * 2, 
			pDestAddr		:= ADR(SlaveCom[SlaveNo]^.Data), 
			bExecute		:= Execute, 
			tTimeout		:= , 
			bBusy			=> StartJob, 
			bError			=> Error, 
			nErrId			=> ErrorID);
	
	ELSIF 	SlaveCom[SlaveNo]^.Jobs[JobNo].FunctionCode = 5 THEN
		WriteSingleCoil(
			sIPAddr			:= SlaveCom[SlaveNo]^.ipAddr, 
			nTCPPort		:= TO_UINT(SlaveCom[SlaveNo]^.Port), 
			nUnitID			:= SlaveCom[SlaveNo]^.Address, 
			nMBAddr			:= SlaveCom[SlaveNo]^.jobs[JobNo].startAddress, 
			nValue			:= SlaveCom[SlaveNo]^.data[1], 
			bExecute		:= Execute, 
			tTimeout		:= , 
			bBusy			=> StartJob, 
			bError			=> Error, 
			nErrId			=> ErrorID);
	
	ELSIF 	SlaveCom[SlaveNo]^.Jobs[JobNo].FunctionCode = 6 THEN
		WriteSingleReg(
			sIPAddr			:= SlaveCom[SlaveNo]^.ipAddr, 
			nTCPPort		:= TO_UINT(SlaveCom[SlaveNo]^.Port), 
			nUnitID			:= SlaveCom[SlaveNo]^.Address, 
			nMBAddr			:= SlaveCom[SlaveNo]^.jobs[JobNo].startAddress, 
			nValue			:= SlaveCom[SlaveNo]^.data[1], 
			bExecute		:= Execute, 
			tTimeout		:= , 
			bBusy			=> StartJob, 
			bError			=> Error, 
			nErrId			=> ErrorID);
			
	ELSIF 	SlaveCom[SlaveNo]^.Jobs[JobNo].FunctionCode = 8 THEN
		Diagnose(
			sIPAddr			:= SlaveCom[SlaveNo]^.ipAddr, 
			nTCPPort		:= TO_UINT(SlaveCom[SlaveNo]^.Port), 
			nUnitID			:= SlaveCom[SlaveNo]^.Address, 
			bExecute		:= Execute, 
			tTimeout		:= , 
			bBusy			=> StartJob, 
			bError			=> Error, 
			nErrId			=> ErrorID);	
			
	ELSIF 	SlaveCom[SlaveNo]^.Jobs[JobNo].FunctionCode = 15 THEN
		WriteCoils(
			sIPAddr			:= SlaveCom[SlaveNo]^.ipAddr, 
			nTCPPort		:= TO_UINT(SlaveCom[SlaveNo]^.Port), 
			nUnitID			:= SlaveCom[SlaveNo]^.Address, 
			nQuantity		:= SlaveCom[SlaveNo]^.jobs[JobNo].Quantity, 
			nMBAddr			:= SlaveCom[SlaveNo]^.jobs[JobNo].startAddress, 
			cbLength		:= SlaveCom[SlaveNo]^.jobs[JobNo].Quantity, 
			pSrcAddr		:= ADR(SlaveCom[SlaveNo]^.Data), 
			bExecute		:= Execute, 
			tTimeout		:= , 
			bBusy			=> StartJob, 
			bError			=> Error, 
			nErrId			=> ErrorID);
	
	ELSIF 	SlaveCom[SlaveNo]^.Jobs[JobNo].FunctionCode = 16 THEN
		WriteRegs(
			sIPAddr			:= SlaveCom[SlaveNo]^.ipAddr, 
			nTCPPort		:= TO_UINT(SlaveCom[SlaveNo]^.Port), 
			nUnitID			:= SlaveCom[SlaveNo]^.Address, 
			nQuantity		:= SlaveCom[SlaveNo]^.jobs[JobNo].Quantity, 
			nMBAddr			:= SlaveCom[SlaveNo]^.jobs[JobNo].startAddress, 
			cbLength		:= SlaveCom[SlaveNo]^.jobs[JobNo].Quantity, 
			pSrcAddr		:= ADR(SlaveCom[SlaveNo]^.Data), 
			bExecute		:= Execute, 
			tTimeout		:= , 
			bBusy			=> StartJob, 
			bError			=> Error, 
			nErrId			=> ErrorID);
			
	ELSIF 	SlaveCom[SlaveNo]^.Jobs[JobNo].FunctionCode = 23 THEN
		// not implemented
(*		ReadWriteRegs(
			sIPAddr			:= SlaveCom[SlaveNo]^.ipAddr, 
			nTCPPort		:= SlaveCom[SlaveNo]^.Port, 
			nUnitID			:= SlaveCom[SlaveNo]^.Address, 
			nReadQuantity	:= SlaveCom[SlaveNo]^.jobs[JobNo].Quantity, 
			nMBReadAddr		:= SlaveCom[SlaveNo]^.jobs[JobNo].startAddress, 
			nWriteQuantity	:= , // missing
			nMBWriteAddr	:= , // missing
			cbDestLength	:= SlaveCom[SlaveNo]^.jobs[JobNo].Quantity, 
			pDestAddr		:= ADR(SlaveCom[SlaveNo]^.Data),
			cbSrcLength		:= , // missing
			pSrcAddr 		:= , // missing
			bExecute		:= Execute, 
			tTimeout		:= , 
			bBusy			=> StartJob, 
			bError			=> Error, 
			nErrId			=> ErrorID);	

*)			
	END_IF
END_METHOD

END_FUNCTION_BLOCK

// ---- POUs/Connectivity/TF625x-Modbus/Master/TF6255-ModbusRtu/ModbusRtuMasterPC.TcPOU
{attribute 'no_check'}
// ModBus comunication master to multible slaves useing RTU protocol
// based on TF6255 - required lib: Tc2_ModbusRTU
FUNCTION_BLOCK ModbusRtuMasterPC
VAR CONSTANT
	MIN_SLAVE												:	INT := 1;
	MAX_SLAVE												:	INT := PARAM.MODBUS_MAX_SLAVES_OF_MASTER;
END_VAR
VAR_INPUT
	Enable													:	BOOL; 			// FB will be processed as long as enable is TRUE 
	ResetTrig												:	BOOL;			// The function block will be reset with a rising edge 
	SlaveCom												:	ARRAY[MIN_SLAVE..MAX_SLAVE] OF POINTER TO ModbusSlaveCom;
	Timestamp												:	DT;
END_VAR         	
VAR_OUTPUT      	
	Error													:	BOOL;			// Rising edge of Error informs that an error occurred during the execution of the Function Block 
	ErrorID													:	MODBUS_ERRORS;	// Error identification 
	ErrorText												:	STRING;
END_VAR
VAR
(* memory **************************************************)
	state 													:	INT := 0;
	JobNo													:	INT := 0;
	SlaveNo													:	INT := 0;
(* trigger *************************************************)

(* timer ***************************************************)

(* blocks **************************************************)
	com														:	ModbusRtuMaster_PcCOM := (Timeout := DEFAULT_ADS_TIMEOUT);
//	com														:	ModbusRtuMaster_KL6x22B := (Timeout := DEFAULT_ADS_TIMEOUT);
//	com														:	ModbusRtuMaster_KL6x5B := (Timeout := DEFAULT_ADS_TIMEOUT);
(* internal used variables *********************************)
	i,j,k													:	INT :=0;

END_VAR

(* ModBus RTU comunication to multible slaves 	JHue V1.0			*)
(* uncomment necessary master funktion block 						*)
(* use TC2_ModBusRTU.lib											*)
(********************************************************************)

	CASE state OF
	0:	(* Idle *)
		IF Enable 
		THEN
			k 												:=	0;
			JobNo  :=  SlaveNo								:=	1;
			state 											:=	10;
		END_IF

	10: 
		IF GetNextSlave() 
		THEN (* find Slave *)
			k 												:= 0;
			IF GetNextJob() 
			THEN (* find JobNo *)
				SlaveCom[SlaveNo]^.currentJobIdx 			:= JobNo;
				SlaveCom[SlaveNo]^.writeJobRequested 		:= SlaveCom[SlaveNo]^.Jobs[JobNo].FunctionCode >= 5;
				State 										:= SEL(SlaveCom[SlaveNo]^.writeJobRequested, 20, 15);
			END_IF
		ELSE
			state 											:=	0;
		END_IF
	
	15: (* wait for valid write date *)
		IF NOT SlaveCom[SlaveNo]^.writeJobRequested
		THEN
			SlaveCom[SlaveNo]^.Jobs[JobNo].Valid 			:= FALSE;
			state 											:= 0;
		END_IF

	20: (* start job *)	
		IF NOT StartJob(FALSE) // Busy
		THEN						
			state 											:= 30;
		END_IF

	30: (* wait for com cycle *)
		IF NOT StartJob(TRUE) THEN // Busy
			IF Error 
			THEN
				ErrorText									:= CONCAT('Error at SlaveNo: ',	CONCAT(INT_TO_STRING(SlaveNo), CONCAT(', JobNo: ', INT_TO_STRING(JobNo))));
				SlaveCom[SlaveNo]^.countBad 				:= SlaveCom[SlaveNo]^.countBad +1;
				state 										:= 98; 
			ELSE
				SlaveCom[SlaveNo]^.countGood 				:= SlaveCom[SlaveNo]^.countGood +1;
				SlaveCom[SlaveNo]^.Jobs[JobNo].Valid 		:= TRUE;
				SlaveCom[SlaveNo]^.Jobs[JobNo].TimeStamp 	:= Timestamp;
				JobNo 										:= JobNo + 1;
				state 										:= 10;	(* next job *)
			END_IF
			StartJob(FALSE);
		END_IF

	98: (* wait for quit *)
		IF ResetTrig THEN
			reset();
		END_IF

	END_CASE

METHOD PRIVATE getNextJob : Bool
VAR_INPUT
END_VAR
	
	WHILE SlaveCom[SlaveNo]^.Jobs[JobNo].FunctionCode = 0 DO
		JobNo 											:= JobNo + 1;
		IF JobNo > SlaveCom[SlaveNo]^.MAX_SLAVE_JOB THEN
			JobNo 										:= SlaveCom[SlaveNo]^.MIN_SLAVE_JOB;
			SlaveNo 									:= SlaveNo + 1;
			GetNextJob									:= FALSE;
			RETURN;
		END_IF
	END_WHILE
	GetNextJob											:= TRUE;
END_METHOD

METHOD PRIVATE getNextSlave : Bool
VAR_INPUT
END_VAR
	WHILE SlaveCom[SlaveNo] = 0 or_else not SlaveCom[SlaveNo]^.Enable DO
		SlaveNo 										:= SlaveNo + 1;
		IF SlaveNo > MAX_SLAVE 
		THEN
			k 											:= k + 1;
			SlaveNo 									:= MIN_SLAVE;
		ELSIF k = 2 
		THEN
			k 											:= 0;
			GetNextSlave								:= FALSE;
			RETURN;
		END_IF	
	END_WHILE
	GetNextSlave										:= TRUE;
END_METHOD

METHOD PUBLIC reset : BOOL //Return value = TRUE if execution finished
VAR_INPUT
END_VAR
IF State = 98 
THEN
	Error													:= FALSE;
	ErrorID													:= 0;
	ErrorText												:= '';
	state													:= 0;
END_IF
reset													:= TRUE;
END_METHOD

METHOD PRIVATE startJob : BOOL //Return value = TRUE if busy - TRUE as long as the job is busy
VAR_INPUT
	Execute							: BOOL;
END_VAR
(* ModbusCOM Baustein mit parametern antriggern *)
	IF 		SlaveCom[SlaveNo]^.Jobs[JobNo].FunctionCode = 1 THEN
		com.ReadCoils(
			UnitID			:= SlaveCom[SlaveNo]^.Address,				(*UnitID: Modbus Stationsadresse (1..247). Der Modbus-Slave antwortet nur, wenn er Telegramme mit seiner eigenen Stationsadresse empfängt. optional können hier auch Sammeladressen eingestellt werden um auf beliebige Anfragen zu antworten. Die Adresse 0 ist für Broadcast-Telegramme reserviert und somit keine gültige Stationsadresse.*)
			Quantity		:= SlaveCom[SlaveNo]^.jobs[JobNo].Quantity,		(*Quantity: Anzahl der zu lesenden oder zu schreibenden Datenworte bei Wort-orientierten Modbus-Funktionen. Bei Bit-orientierten Modbus-Funktionen gibt Quantity die Anzahl der Bits (Inputs oder Coils) an.*)
			MBAddr			:= SlaveCom[SlaveNo]^.jobs[JobNo].startAddress,	(*MBAddr: Modbus-Datenadresse, von der die Daten aus dem Endgerät (Slave) gelesen werden. Diese Adresse wird unverändert zum Slave übertragen und wird dort als Datenadresse interpretiert.*)
			cbLength		:= SlaveCom[SlaveNo]^.jobs[JobNo].Quantity, 	(*cbLength : Größe der verwendeten Datenvariable für Sende- oder Lese-Aktionen in Bytes. cbLength muss größer oder gleich der durch Quantity bestimmten übertragenen Datenmenge sein. Bei Wortzugriffen gilt z. B.: [cbLength >= Quantity * 2]. cbLength kann mit SIZEOF(ModbusDaten) berechnet werden.*)
			pMemoryAddr		:= ADR(SlaveCom[SlaveNo]^.Data),				(*pMemoryAddr: Speicheradresse in der SPS, die mit ADR(ModbusDaten) berechnet wird. Bei Leseaktionen werden die gelesenen Daten in der adressierten Variablen abgelegt. Bei Sende-Aktionen werden die Daten aus der adressierten Variablen zum Endgerät übertragen.*)
			Execute			:= Execute,
			Timeout			:= ,
			BUSY			=> StartJob,									(*Busy: Zeigt an, dass der Funktionsbaustein aktiv ist. Busy wird mit steigender Flanke an Execute TRUE und wird wieder FALSE nachdem die gestartete Aktion beendet ist. Es kann immer nur eine Aktion gleichzeitig aktiv sein.*)
			Error			=> Error,										(*Error: Zeigt an, dass bei der Bearbeitung einer Aktion ein Fehler aufgetreten ist*)
			ErrorId			=> ErrorID);									(*ErrorId: Zeigt eine Fehlernummer im Falle einer gestörten oder fehlerhaften Kommunikation an.*)	
	
	ELSIF 	SlaveCom[SlaveNo]^.Jobs[JobNo].FunctionCode = 3 THEN
		com.ReadRegs(
			UnitID			:= SlaveCom[SlaveNo]^.Address,		
			Quantity		:= SlaveCom[SlaveNo]^.jobs[JobNo].Quantity,
			MBAddr			:= SlaveCom[SlaveNo]^.jobs[JobNo].startAddress,
			cbLength		:= SlaveCom[SlaveNo]^.jobs[JobNo].Quantity * 2,
			pMemoryAddr		:= ADR(SlaveCom[SlaveNo]^.data),
			Execute			:= Execute,
			Timeout			:= ,
			BUSY			=> StartJob,
			Error			=> Error,
			ErrorId			=> ErrorID);
	
	ELSIF 	SlaveCom[SlaveNo]^.Jobs[JobNo].FunctionCode = 4 THEN
		com.ReadInputRegs(
			UnitID			:= SlaveCom[SlaveNo]^.Address,		
			Quantity		:= SlaveCom[SlaveNo]^.jobs[JobNo].Quantity,
			MBAddr			:= SlaveCom[SlaveNo]^.jobs[JobNo].startAddress,
			cbLength		:= SlaveCom[SlaveNo]^.jobs[JobNo].Quantity * 2,
			pMemoryAddr		:= ADR(SlaveCom[SlaveNo]^.data),
			Execute			:= Execute,
			Timeout			:= ,
			BUSY			=> StartJob,
			Error			=> Error,
			ErrorId			=> ErrorID);
	
	ELSIF 	SlaveCom[SlaveNo]^.Jobs[JobNo].FunctionCode = 5 THEN
		com.WriteSingleCoil(
			UnitID			:= SlaveCom[SlaveNo]^.Address,		
			Quantity		:= SlaveCom[SlaveNo]^.jobs[JobNo].Quantity,
			MBAddr			:= SlaveCom[SlaveNo]^.jobs[JobNo].startAddress,
			cbLength		:= SlaveCom[SlaveNo]^.jobs[JobNo].Quantity,
			pMemoryAddr		:= ADR(SlaveCom[SlaveNo]^.data),
			Execute			:= Execute,
			Timeout			:= ,
			BUSY			=> StartJob,
			Error			=> Error,
			ErrorId			=> ErrorID);
			
	ELSIF 	SlaveCom[SlaveNo]^.Jobs[JobNo].FunctionCode = 6 THEN
		com.WriteSingleRegister(
			UnitID			:= SlaveCom[SlaveNo]^.Address,		
			Quantity		:= SlaveCom[SlaveNo]^.jobs[JobNo].Quantity,
			MBAddr			:= SlaveCom[SlaveNo]^.jobs[JobNo].startAddress,
			cbLength		:= SlaveCom[SlaveNo]^.jobs[JobNo].Quantity,
			pMemoryAddr		:= ADR(SlaveCom[SlaveNo]^.data),
			Execute			:= Execute,
			Timeout			:= ,
			BUSY			=> StartJob,
			Error			=> Error,
			ErrorId			=> ErrorID);
		
	ELSIF 	SlaveCom[SlaveNo]^.Jobs[JobNo].FunctionCode = 8 THEN
		com.Diagnostics(
			UnitID			:= SlaveCom[SlaveNo]^.Address,		
			Quantity		:= SlaveCom[SlaveNo]^.jobs[JobNo].Quantity,
			MBAddr			:= SlaveCom[SlaveNo]^.jobs[JobNo].startAddress,
			cbLength		:= SlaveCom[SlaveNo]^.jobs[JobNo].Quantity,
			pMemoryAddr		:= ADR(SlaveCom[SlaveNo]^.data),
			Execute			:= Execute,
			Timeout			:= ,
			BUSY			=> StartJob,
			Error			=> Error,
			ErrorId			=> ErrorID);
	
	ELSIF 	SlaveCom[SlaveNo]^.Jobs[JobNo].FunctionCode = 15 THEN
		com.WriteMultipleCoils(
			UnitID			:= SlaveCom[SlaveNo]^.Address,		
			Quantity		:= SlaveCom[SlaveNo]^.jobs[JobNo].Quantity,
			MBAddr			:= SlaveCom[SlaveNo]^.jobs[JobNo].startAddress,
			cbLength		:= SlaveCom[SlaveNo]^.jobs[JobNo].Quantity,
			pMemoryAddr		:= ADR(SlaveCom[SlaveNo]^.data),
			Execute			:= Execute,
			Timeout			:= ,
			BUSY			=> StartJob,
			Error			=> Error,
			ErrorId			=> ErrorID);
	
	ELSIF 	SlaveCom[SlaveNo]^.Jobs[JobNo].FunctionCode = 16 THEN
		com.WriteRegs(
			UnitID			:= SlaveCom[SlaveNo]^.Address,		
			Quantity		:= SlaveCom[SlaveNo]^.jobs[JobNo].Quantity,
			MBAddr			:= SlaveCom[SlaveNo]^.jobs[JobNo].startAddress,
			cbLength		:= SlaveCom[SlaveNo]^.jobs[JobNo].Quantity,
			pMemoryAddr		:= ADR(SlaveCom[SlaveNo]^.data),
			Execute			:= Execute,
			Timeout			:= ,
			BUSY			=> StartJob,
			Error			=> Error,
			ErrorId			=> ErrorID);	
	END_IF
END_METHOD

END_FUNCTION_BLOCK

// ---- POUs/Connectivity/TF6310-TcpServer/UdpBasic/UDPSendRecCtrl.TcPOU
{attribute 'no_check'}
//Send or receive data via TCP connection 
//based on TF6310, required lib: Tc2_TcpIp - see Beckhoff Infosys for more information
FUNCTION_BLOCK UDPSendRecCtrl Extends FbBase
VAR_OUTPUT CONSTANT
	FNC_RECEIVE												:	INT := 0;
	FNC_SEND												:	INT := 1;
END_VAR             										
VAR_INPUT           										
	Fnc														:	INT (FNC_RECEIVE..FNC_SEND) := FNC_RECEIVE;
{attribute 'displaymode':='binary'}
	Options													:	BYTE := 2#0000_0000; // Options Bit .0 = Do NOT restart receive intern / Receive intern nicht neustarten
	SrvNetId												: 	T_AmsNetId := ''; 	// server ams net id
	RemoteHost 												: 	T_IPv4Addr; // Target ip adress - only for send data *)
	RemotePort												: 	UDINT; 	// target port - only for send data *)
	Timeout													: 	TIME := DEFAULT_ADS_TIMEOUT; //ADS timeout
	hSocket													:	T_HSOCKET; 	// Socket handle provided by Server/Handle
	pData													:	POINTER TO BYTE; 	//Pointer do send/res data field 
	cbData													:	UDINT; 	// Size of send/rec data field 
	EnableDebugMode											:	BOOL;	// Write debug information into twincat logger
END_VAR
VAR_OUTPUT
	RecBytes 												:  UDINT;  	// Count of received bytes
	WinsockErrorId											:	E_WinsockError; //Winsocket error enum - see TF6310 documentation for further information
	RecRemoteHost 											:  STRING(15); 	// Remote host IP
	RecRemotePort											:  UDINT; 	// Remote host port
END_VAR                 									
VAR                     	
(* cache ************************************************************)
	MemFnc													:	INT := -1;

(* function-block instances ***************************************************************)
	SocketSend												:	FB_SocketUdpSendTo;
	SocketReceive											:	FB_SocketUdpReceiveFrom;

END_VAR


(* Execute ***************************************************************************************)
	rtExecute(CLK := Execute);
	IF rtExecute.Q
		AND MemFnc < 0
	THEN
		MemFnc 												:= SEL(Fnc = FNC_SEND, FNC_RECEIVE , FNC_SEND) ;
		Busy												:= TRUE;
		Done												:= FALSE;
		Error												:= FALSE;
		ErrorID												:= 0;
	END_IF

(* Call Method ***********************************************************************************)
	CASE MemFnc OF
	FNC_SEND:
		SEND( Execute := Execute);

	FNC_RECEIVE:
		Receive( Execute := Execute);
			
	-1:
		IF NOT Execute
		THEN
			Busy											:= FALSE;
			Done											:= FALSE;
			Error											:= FALSE;
			ErrorID											:= 0;
		END_IF                              				
	ELSE                                    				
		Busy												:= FALSE;
		Done												:= FALSE;
		Error												:= Execute;
		ErrorID												:= E_AdsErr.DEVICE_INVALIDPARM;
	END_CASE                                	
                                            	
(*************************************************************************************************)

PROPERTY PUBLIC optDoNotRestartReceiveCylic : BOOL
GET
optDoNotRestartReceiveCylic := Options.0;
END_GET
SET
Options.0 := optDoNotRestartReceiveCylic;
END_SET
END_PROPERTY

METHOD PUBLIC receive : BOOL	//Return value = TRUE if busy
//required parameter
//hSocket
//pData
//cbData
VAR_INPUT
	Execute													:	BOOL;
END_VAR
	MemFnc													:= FNC_RECEIVE;
	THIS^.Execute											:= Execute;
	
IF pData = 0 
THEN
	Busy													:= NOT Error;
	Error													:= TRUE;
	ErrorId													:= E_AdsErr.DEVICE_INVALIDPARM;
	Done													:= FALSE;
	MemFnc													:= SEL(Execute , -1 ,MemFnc); 
	RETURN;
END_IF

	IF Execute
	THEN
		Error												:=	FALSE;
		ErrorId												:= 0;
		SocketReceive.bExecute 								:= TRUE;
	ELSIF NOT SocketReceive.bBusy       					
	THEN                                					
		Error												:=	FALSE;
		ErrorId												:= 0;
		SocketReceive.bExecute 								:= FALSE;
	END_IF

	SocketReceive(
		sSrvNetId	:= SrvNetId,
		hSocket		:= hSocket,
		cbLen		:= cbData,
		pDest		:= pData,
		bExecute	:= ,
		tTimeout	:= Timeout,
		bBusy		=> Busy,
		bError		=> ,
		nErrId		=> ,
		nRecBytes	=> );

	IF NOT SocketReceive.bBusy
		AND NOT SocketReceive.bError
		AND SocketReceive.bExecute
	THEN
		IF EnableDebugMode
			AND SocketReceive.nRecBytes > 0
			AND NOT Done
		THEN
			hSocket.remoteAddr.sAddr						:= SocketReceive.sRemoteHost;
			hSocket.remoteAddr.nPort						:= SocketReceive.nRemotePort;
			ADSLOGDINT(	ADSLOG_MSGTYPE_ERROR OR ADSLOG_MSGTYPE_LOG, CONCAT('%d Bytes received / ', HSOCKET_TO_STRING(hSocket)) , UDINT_TO_DINT(SocketReceive.nRecBytes));
		END_IF
		Done												:= SocketReceive.nRecBytes > 0 OR Options.0; (* Done melden nach jedenm Lesezyklus, egal ob Daten empfangen wurden *)
		IF NOT Done
		THEN (* Nur Done melden wenn auch was empfangen wurde *)
			SocketReceive(bExecute := FALSE);
			SocketReceive(bExecute := TRUE, bBusy => Busy);
		END_IF
		RecBytes											:= SEL(Done , 0 ,SocketReceive.nRecBytes);
	ELSE                                					
		Done												:= FALSE;
	END_IF                              	

	IF NOT Busy
	THEN
		IF SocketReceive.bExecute
		THEN
			Error											:=	SocketReceive.bError;
			IF SocketReceive.nErrId >= 16#80070000
			THEN
				ErrorId										:= E_AdsErr.CLIENT_W32ERROR;
				WinsockErrorId								:= ADSERROR_TO_WSERROR(SocketReceive.nErrId);
			ELSE                    						
				ErrorId										:= SocketReceive.nErrId;
				WinsockErrorId								:= WSOK;
			END_IF                  						
		END_IF                      	
		IF NOT Execute
		THEN
			MemFnc											:= -1;
			SocketReceive(bExecute := FALSE);
		END_IF
	END_IF
	
	//Method return
	Receive													:= Busy;
END_METHOD

METHOD PUBLIC send : BOOL 	//Return value = TRUE if busy
//required parameter
//hSocket
//pData
//cbData
//RemoteHost
//RemotePort
VAR_INPUT
	Execute													:	BOOL;
END_VAR
	MemFnc													:= FNC_SEND;
	THIS^.Execute											:= Execute;
	                                    					
IF pData = 0 THEN                       					
	Busy													:= NOT Error;
	Error													:= TRUE;
	ErrorId													:= E_AdsErr.DEVICE_INVALIDPARM;
	Done													:= FALSE;
	MemFnc													:= SEL(Execute , -1 ,MemFnc); 
	RETURN;
END_IF

	IF Execute
	THEN
		Error												:= FALSE;
		ErrorId												:= 0;
		SocketSend.bExecute 								:= TRUE;
	ELSIF NOT SocketSend.bBusy          					
	THEN                                					
		Error												:= FALSE;
		ErrorId												:= 0;
		SocketSend.bExecute 								:= FALSE;
	END_IF                              	
	
	SocketSend(
		sSrvNetId	:= SrvNetId,
		hSocket		:= hSocket,
		sRemoteHost	:= RemoteHost,
		nRemotePort	:= RemotePort,
		cbLen		:= cbData,
		pSrc		:= pData,
		bExecute	:= ,
		tTimeout	:= Timeout,
		bBusy		=> Busy,
		bError		=> ,
		nErrId		=> );

	IF NOT SocketSend.bBusy
		AND NOT SocketSend.bError
		AND SocketSend.bExecute
	THEN
		IF NOT Done
			AND EnableDebugMode
		THEN
			hSocket.remoteAddr.sAddr						:= SocketSend.sRemoteHost;
			hSocket.remoteAddr.nPort						:= SocketSend.nRemotePort;
			ADSLOGDINT(	ADSLOG_MSGTYPE_ERROR OR ADSLOG_MSGTYPE_LOG, CONCAT('%d Bytes sended / ', HSOCKET_TO_STRING(hSocket)) , UDINT_TO_DINT(cbData));
		END_IF
		Done												:= TRUE;
	ELSE                                					
		Done												:= FALSE;
	END_IF                              	
                                        	
	IF NOT Busy
	THEN
		IF SocketSend.bExecute
		THEN
			Error											:=	SocketSend.bError;
			IF SocketSend.nErrId >= 16#80070000
			THEN
				ErrorId										:= E_AdsErr.CLIENT_W32ERROR;
				WinsockErrorId								:= ADSERROR_TO_WSERROR(SocketSend.nErrId);
			ELSE                    						
				ErrorId										:= SocketSend.nErrId;
				WinsockErrorId								:= WSOK;
			END_IF                  	
		END_IF
		IF NOT Execute
		THEN
			MemFnc											:= -1;
			SocketSend(bExecute := FALSE);
		END_IF
	END_IF
	
	//Method return
	Send													:= Busy;
END_METHOD

END_FUNCTION_BLOCK

// ---- POUs/ControllerTools/PT1Filter.TcPOU
//Low pass filter with a programmable time Tn and factor Kp.
FUNCTION_BLOCK PT1Filter
VAR_INPUT
	Enable													:	BOOL ; 	// FB will be processed as long as enable is TRUE 
	In														:	LREAL := 0.0;	// Actual value
	ResetTrig												:	BOOL ; 	// The function block will be reset with a rising edge 
	Sync													:	BOOL ; 	// Synchronise In to Q - equivalent to Synchronize method
	Kp														:	LREAL := 1.0; 	// Gain
	Tn														:	TIME := T#1S; 	// Integral time 
	Cycletime 												:	TIME := T#10MS;	// cycletime 
END_VAR	            										
VAR_OUTPUT          										
	Q														: LREAL;			// Output
	Error													: BOOL;				// Rising edge of Error informs that an error occurred during the execution of the Function Block 
END_VAR             										
VAR                 	
	Q_old													: LREAL;
END_VAR

(**************************************************************************************
	formula: 
	y(k) = [1-T/T1]	* y(k-1)
			+ T/T1		* v 		* e(k) 
*************************************************************************************)

	Error 													:= Cycletime = T#0MS OR  tn = T#0MS OR Kp = 0.0;
                            								
	IF Enable               								
		AND NOT Error       								
	THEN                    								
		Q 													:=  (1- TIME_TO_LREAL(Cycletime) / TIME_TO_LREAL(Tn))	* Q_old
															 	+ TIME_TO_LREAL(Cycletime) / TIME_TO_LREAL(Tn)	* Kp		* In;
		Q_Old 												:= Q;
	ELSE //Hold
		;
	END_IF

	IF ResetTrig
	THEN
		reset();
	ELSIF Sync
	THEN
		Synchronize(IN);
	END_IF

(************************************************************************************)

METHOD reset : BOOL //Return value = TRUE if execution finished
VAR_INPUT
END_VAR
Q := Q_old 				:= 0.0;
reset				:= TRUE;
END_METHOD

METHOD PUBLIC synchronize : BOOL //Return value = TRUE if execution finished
VAR_INPUT
	IN						:	LREAL;
END_VAR
Q 	:= Q_Old 	 := IN;
Synchronize		:= TRUE;
END_METHOD

END_FUNCTION_BLOCK

// ---- POUs/DataBuffer/Ringbuffer/RingbufferExt.TcPOU
//Ringbuffer extended with dynamical allocation of memory 
{attribute 'enable_dynamic_creation'}
FUNCTION_BLOCK RingbufferExt EXTENDS RingbufferBase
VAR_OUTPUT CONSTANT
END_VAR   
VAR_INPUT
	MaxNoOfEntrys											: 	UDINT := 10;	//0 = dynamically allocation / <> 0 = pre allcoation of memory based on size of first entry (n * data size) 
END_VAR
VAR_OUTPUT
	pMemory													: 	POINTER TO BYTE := 0;	//start address of buffer data
	SizeOfMemory											: 	UDINT := 0;	//size of buffer
END_VAR
VAR
	MemSizeAllocatedMemory									:	UDINT := 0; //Allocated memory 
	MemSizeOfData											:	UDINT;
	MemMaxNoOfEntrys										:	UDINT;
	ExtInterlock											:	BOOL;
END_VAR

;

METHOD PROTECTED FINAL allocate : BOOL
VAR_IN_OUT
	SizeOfData												:	UDINT;
END_VAR
VAR
	pDummy													:	POINTER TO BYTE;	
End_Var
IF pMemory = 0
THEN
	IF SizeOfData = 0 OR MaxNoOfEntrys = 0
	THEN
		Allocate											:= FALSE;	
	ELSE
		MemSizeOfData										:= SizeOfData;
		MemMaxNoOfEntrys									:= MaxNoOfEntrys;
		SizeOfMemory										:= MemSizeOfData * MemMaxNoOfEntrys;
		MemSizeAllocatedMemory								:= SizeOfMemory;
		pMemory												:= __NEW(BYTE,SizeOfMemory );
		
		IF PARAM.ENABLE_DEBUG_MSG_DYNAMIC_MEM_ALLOCATION
		THEN
			AdsLogHint('EngineeringToolbox | FB FifoExt | An instance allocated %s bytes from the dynamic memory of the ADS router memory pool', TO_STRING(SizeOfMemory));
		END_IF
	END_IF

ELSIF SizeOfData = MemSizeOfData AND MaxNoOfEntrys = MemMaxNoOfEntrys
THEN
	Allocate												:= TRUE;
	
ELSIF SizeOfData > MemSizeOfData OR MaxNoOfEntrys > MemMaxNoOfEntrys
THEN //Since increased, allocate new memory
	MemSizeAllocatedMemory									:= SizeOfData * MaxNoOfEntrys;
	pDummy													:= __NEW(BYTE, MemSizeAllocatedMemory); 
	
	 //Size of data still the same, copy old data to reuse
	IF MemSizeOfData = SizeOfData AND Count > 0
	THEN
		MEMCPY(pDummy,pMemory, SizeOfMemory);
	END_IF
	
	//Copy new settings to local variales
	MemSizeOfData											:= SizeOfData;
	MemMaxNoOfEntrys										:= MaxNoOfEntrys;	
	SizeOfMemory 											:= MemSizeAllocatedMemory;

	__DELETE(pMemory);  //Delete reference to old memory
	pMemory													:= pDummy; //Take over new pointer to new memory
	
	IF PARAM.ENABLE_DEBUG_MSG_DYNAMIC_MEM_ALLOCATION
	THEN
		AdsLogWarn('EngineeringToolbox | FB FifoExt | Value of "MaxNoOfEntrys" or data size increased and one instance allocated additional %s bytes from the dynamic memory of the ADS router memory pool', TO_STRING(SizeOfMemory));
	END_IF
	
	Allocate												:= TRUE;
	
ELSE //Size decreased
	IF MemSizeOfData <> SizeOfData AND Count > 0
	THEN //Size of data changed, erease memory 
		MEMSET(pMemory,0, MemSizeAllocatedMemory);
	ELSE //Size of data the same, keep current data
		;
	END_IF
	
	//Copy new settings to local variales
	MemSizeOfData											:= SizeOfData;
	MemMaxNoOfEntrys										:= MaxNoOfEntrys;
	SizeOfMemory											:= MemSizeOfData * MemMaxNoOfEntrys;
	Allocate												:= TRUE;
END_IF
END_METHOD

METHOD PUBLIC dequeue : BOOL //TRUE if method was successful
VAR_INPUT
	pData													:	POINTER TO BYTE;	
END_VAR
VAR
END_VAR
Dequeue := SUPER^._Dequeue(pData,SizeOfEntry,This^.pMemory,This^.SizeOfMemory);
END_METHOD

METHOD PUBLIC dequeueStream : BOOL //TRUE if method was successful
VAR_INPUT
	pData													:	POINTER TO BYTE;	
	SizeOfStream											:	UDINT ; //Not greater than SizeOfMemory
END_VAR
VAR
END_VAR
DequeueStream := SUPER^._DequeueStream(pData,SizeOfStream , This^.pMemory,This^.SizeOfMemory);
END_METHOD

METHOD PUBLIC enqueue : BOOL //TRUE if method was successful
VAR_INPUT
	pData													:	POINTER TO BYTE;
	SizeOfData												:	UDINT;
END_VAR
VAR
END_VAR
IF TestAndSet(ExtInterlock) 
THEN	
	if Allocate(SizeOfData)
	then
		Enqueue 											:= SUPER^._Enqueue(pData,SizeOfData,THIS^.pMemory,THIS^.SizeOfMemory);
		ExtInterlock										:= FALSE;
	else
		Enqueue												:= FALSE;
	END_IF	
ELSE
	Enqueue													:= FALSE;
END_IF
END_METHOD

METHOD PUBLIC enqueueStream : BOOL //TRUE if method was successful
VAR_INPUT
	pData													:	POINTER TO BYTE;
	SizeOfData												:	UDINT; //Size of one entry
	SizeOfStream											:	UDINT ; //Not greater than SizeOfMemory
END_VAR
VAR
END_VAR
IF TestAndSet(ExtInterlock) 
THEN	
	if Allocate(SizeOfData)
	then
		EnqueueStream 										:= SUPER^._EnqueueStream(pData,SizeOfData,SizeOfStream,THIS^.pMemory,THIS^.SizeOfMemory);
		ExtInterlock										:= FALSE;
	else
		EnqueueStream										:= FALSE;
	END_IF	
ELSE
	EnqueueStream											:= FALSE;
END_IF
END_METHOD

METHOD FB_exit : BOOL
VAR_INPUT
	bInCopyCode : BOOL; // if TRUE, the exit method is called for exiting an instance that is copied afterwards (online change).
END_VAR
IF NOT bInCopyCode AND pMemory <> 0
THEN //Release memory in case the PLC stopps
	__DELETE(pMemory);
	SizeOfMemory								:= 0;
END_IF
END_METHOD

//Reset complete ring buffer
METHOD PUBLIC reset : BOOL //TRUE if method is finnished
VAR_INPUT
END_VAR
IF pMemory = 0
THEN //no memroy allocated
	reset													:= TRUE;
ELSE //Just delte the memory
	reset 													:= SUPER^._reset(THIS^.pMemory,THIS^.SizeOfMemory);	
END_IF
END_METHOD

END_FUNCTION_BLOCK

// ---- POUs/EventLogger/getEventClassPriority.TcPOU
{attribute 'no_check'}
//Returns configured level to corresponding event class (see library Param) 
FUNCTION getEventClassPriority : UINT
VAR_INPUT
	TcEventClass											:	E_TcEventClass;
END_VAR
VAR
END_VAR

	CASE tcEventClass OF
	Tc2_System.TCEVENTCLASS_NONE:			GetEventClassPriority	:= PARAM.EVENT_HANDLING_CONFIG.CLASS_NONE_PRIORITY;	
	Tc2_System.TCEVENTCLASS_MAINTENANCE:	GetEventClassPriority	:= PARAM.EVENT_HANDLING_CONFIG.CLASS_MAINTENANCE_PRIORITY;		
	Tc2_System.TCEVENTCLASS_MESSAGE:		GetEventClassPriority	:= PARAM.EVENT_HANDLING_CONFIG.CLASS_MESSAGE_PRIORITY;			
	Tc2_System.TCEVENTCLASS_HINT:			GetEventClassPriority	:= PARAM.EVENT_HANDLING_CONFIG.CLASS_HINT_PRIORITY;	
	Tc2_System.TCEVENTCLASS_STATEINFO:		GetEventClassPriority	:= PARAM.EVENT_HANDLING_CONFIG.CLASS_STATEINFO_PRIORITY;	
	Tc2_System.TCEVENTCLASS_INSTRUCTION:	GetEventClassPriority	:= PARAM.EVENT_HANDLING_CONFIG.CLASS_INSTRUCTION_PRIORITY;	
	Tc2_System.TCEVENTCLASS_WARNING:		GetEventClassPriority	:= PARAM.EVENT_HANDLING_CONFIG.CLASS_WARNING_PRIORITY;	
	Tc2_System.TCEVENTCLASS_ALARM:			GetEventClassPriority	:= PARAM.EVENT_HANDLING_CONFIG.CLASS_ALARM_PRIORITY;	
	Tc2_System.TCEVENTCLASS_PARAMERROR:		GetEventClassPriority	:= PARAM.EVENT_HANDLING_CONFIG.CLASS_PARAMERROR_PRIORITY;		
	ELSE
		GetEventClassPriority										:= PARAM.EVENT_HANDLING_CONFIG.CLASS_ALARM_PRIORITY;
	END_CASE

END_FUNCTION

// ---- POUs/Fieldbus/Profibus/ProfibusMasterDiag.TcPOU
{attribute 'no_check'}
FUNCTION_BLOCK ProfibusMasterDiag
VAR_INPUT                               					
	Enable													:	BOOL := FALSE;		//FB will be processed as long as enable is TRUE 	
	ResetTrig													:	BOOL := FALSE;		//Resets error with rising edge 
	SourceId												:	UDINT := 103020; 	//default
END_VAR                                 	
VAR_OUTPUT                              	
	IO														:	ProfiBusMasterIO;
END_VAR
VAR
(* trigger ********************************************************)
		
(* events *********************************************************)
	EventMasterError										:	EventHandling;
	EventNoteError											:	ARRAY[1..PARAM.PROFIBUS_MASTER_DEV_IO_MAX_SLAVES] OF EventHandling;
(* function-block *************************************************)
	
(* dummy **********************************************************)	
	i														:	INT;
END_VAR

	(* ProfiBus master diagnosis for EL6731 and slaves	V2.0	*)
	(************************************************************)

(* Work IO ***********************************************)
	IO();

(* Master error ******************************************************)
	EventMasterError(
		Flag			:= IO.Error <> 0 AND Enable,
		ConfirmTrig		:= ResetTrig OR NOT Enable,
		MsgId			:= 1,
		SourceId		:= SourceId,
		eClass			:= ,
		Text1			:= ,
		Text2			:= USINT_TO_STRING(IO.Error),
		pText3			:= ADR(IO.Name),
		State			=> );
		
(* Slave note error **************************************)
	FOR i := IO.MIN_SLAVES TO IO.MAX_SLAVES DO		
		EventNoteError[i](
			Flag		:= IO.SlaveDpStates[i] <> 0 AND Enable,
			ConfirmTrig := ResetTrig OR NOT Enable,
			MsgId		:= TO_UINT(i + 1),
			Text1		:= TO_STRING(i),
			Text2		:= TO_STRING(IO.SlaveDpStates[i]),
			pText3		:= ADR(IO.Name),
			SourceId	:= );
		
 	END_FOR
	

		
(*********************************************************)

END_FUNCTION_BLOCK

// ---- POUs/Fieldbus/Profinet/ProfinetControllerIO_wEvents.TcPOU
{attribute 'no_check'}
//EL6631 Profinet Controller IOs via EtherCAT
FUNCTION_BLOCK ProfinetControllerIO_wEvents EXTENDS ProfinetControllerIO
VAR_OUTPUT CONSTANT

END_VAR
VAR_INPUT
	Enable													:	BOOL := FALSE;
	ResetTrig												:	BOOL := FALSE;
	SourceId												:	UDINT := 103040; (* default *)	
END_VAR
VAR_OUTPUT

END_VAR                     					             	
VAR   
(* trigger ********************************************************)
	
(* events *********************************************************)
	EventControllerError									:	EventHandling;
	EventBoxError											:	ARRAY[1..MAX_BOX] OF EventHandling;
	
(* function-block *************************************************)
	
(* dummy **********************************************************)	
	i														:	INT;    
END_VAR

	(* Profinet controller diagnosis for EL6631	and boxes	V3.0*)
	(************************************************************)

(* Work super ***********************************************)
SUPER^();
	
(* Master error *******************************************)
	EventControllerError(
		Flag				:= PnIoError <> 0 AND Enable,
		ConfirmTrig			:= ResetTrig OR NOT Enable,
		MsgId				:= 1,
		SourceId			:= SourceId,
		eClass				:= ,
		Text1				:= TO_STRING(PnIoError),
		Text2				:= ,
		pText3				:= ADR(DevName),
		State				=> );

(* Box error *********************************************)
	FOR i := MIN_BOX TO MAX_BOX DO
		EventBoxError[i](
			Flag			:= PnIoBoxDiag[i] <> 0 AND Enable,
			ConfirmTrig		:= ResetTrig OR NOT Enable,
			MsgId			:= TO_UINT(i + 1),
			SourceId		:= SourceId,
			eClass			:= ,
			Text1			:= TO_STRING(PnIoBoxDiag[i]),
			Text2			:= TO_STRING(i),
			pText3			:= ADR(DevName),
			State			=> );
 	END_FOR

(*********************************************************)

END_FUNCTION_BLOCK

// ---- POUs/Fieldbus/Profinet/ProfinetDeviceIO.TcPOU
{attribute 'no_check'}
//EL6631-0010 Profinet Device IOs via EtherCAT
// it´s possible to set up multi device for diffrent master
FUNCTION_BLOCK ProfinetDeviceIO EXTENDS EcSlaveInfoDataExt
VAR_OUTPUT CONSTANT
	MIN_BOX													:	INT := 1;
	MAX_BOX													:	INT := PARAM.PROFINET_DEVICE_DEV_IO_MAX_BOX;
																
END_VAR
VAR_INPUT
	PnIoBoxCtrl										AT %Q*	:	ARRAY[MIN_BOX ..MAX_BOX] OF UINT;
END_VAR
VAR_OUTPUT                       				
	AoeNetId										AT %I*	:	AMSNETID;		//Link to master AoeNetID
//Box states	             	
	{attribute 'displaymode':='binary'}
	PnIoBoxState									AT %I*	:	ARRAY[MIN_BOX ..MAX_BOX] OF UINT; //Link to box state
END_VAR                     					             	
VAR       
END_VAR

SUPER^();

END_FUNCTION_BLOCK

// ---- POUs/IO/Analog/AnalogIn.TcPOU
{attribute 'no_check'}
FUNCTION_BLOCK AnalogIn
VAR_INPUT
	MinValue												: 	LREAL 	:= 0.0; //In case of enabled extended range on the terminal, the MinValue has to be set accordingly e.g. -10.7V instead of 1-0.0V as scaling is based on full 16bit
	MaxValue												: 	LREAL 	:= 0.0; //In case of enabled extended range on the terminal, the MaxValue has to be set accordingly e.g. 10.7V instead of 10.0V as scaling is based on full 16bit
	NoOfDigits												: 	INT 	(0..10)	:= 0; 	//number of decimal digits of scaled Q variable 
	OutOnError												:	LREAL 	:= 0.000000000000000001;
{attribute 'displaymode':='binary'}                     	
	Options													:	BYTE  := 2#0000_0000; (* 	.0 = FALSE scale value from 0 <-> 32767 / TRUE scale value with sign -32768 <-> 32767
																							.4 = FALSE scale value min -32768 / TRUE scale value to -7629 -> Extended Range Mode of e.g. 4-20mA where 0mA is equel -7629 *)
																							
	Offset													:	LREAL := 0.0;
END_VAR                 									
VAR                                                     	
END_VAR                                                 	
VAR_OUTPUT                                              	
	Q														:	LREAL;		//Scaled result value
	In											AT  %I* 	: 	INT; 		//Hardware Input

{attribute 'displaymode':='binary'}                     	
	Status										AT  %I*		:	WORD := 2#0000_0000_0000_0000; //Terminal status word -> can also be linked with status byte 

END_VAR
VAR
END_VAR

(* read analog value 																					    *)
(* resolution process image			e.g.							/ 0V = 0 / 10V = 32767 / -10V = - 32768 *)
(* or directly with NoOfDigits																	250 -> 25.0°*)
(************************************************************************************************************)
	
